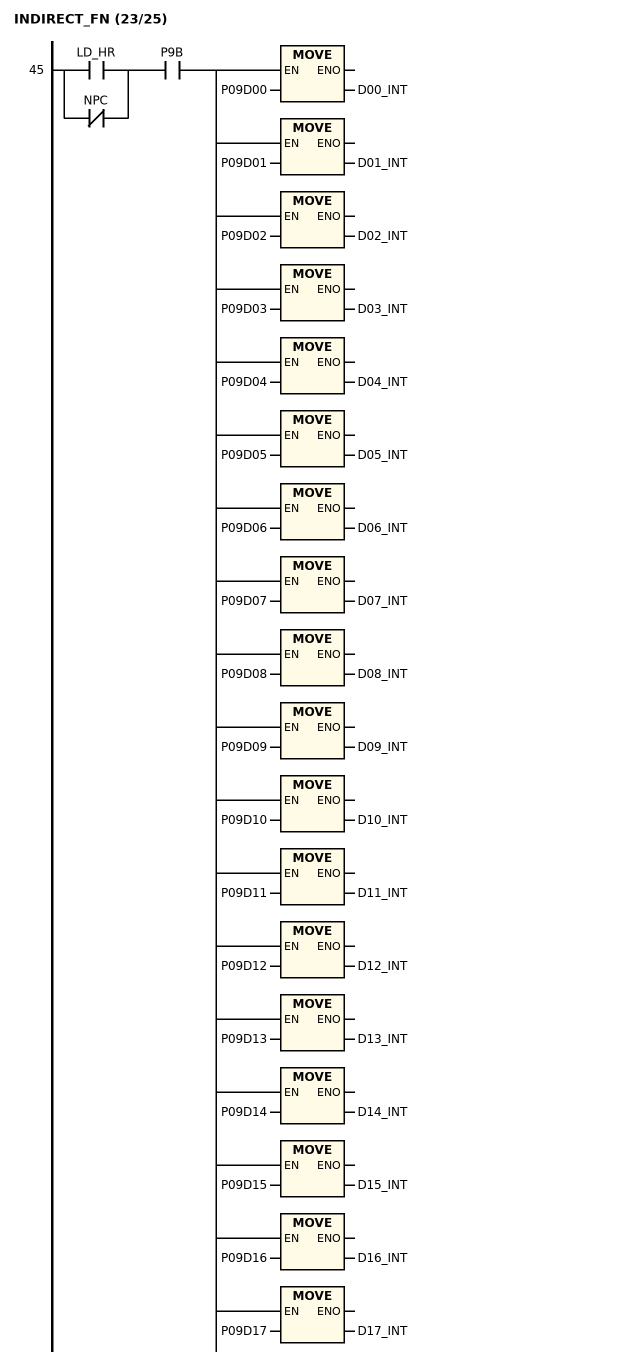
[picture p72: INDIRECT_FN (LD)]
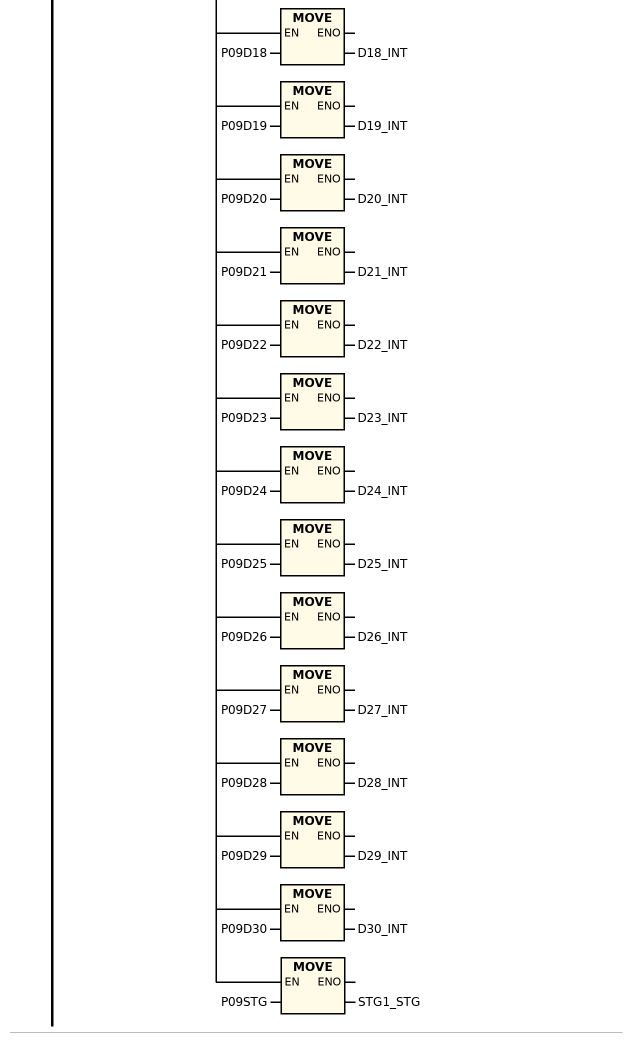
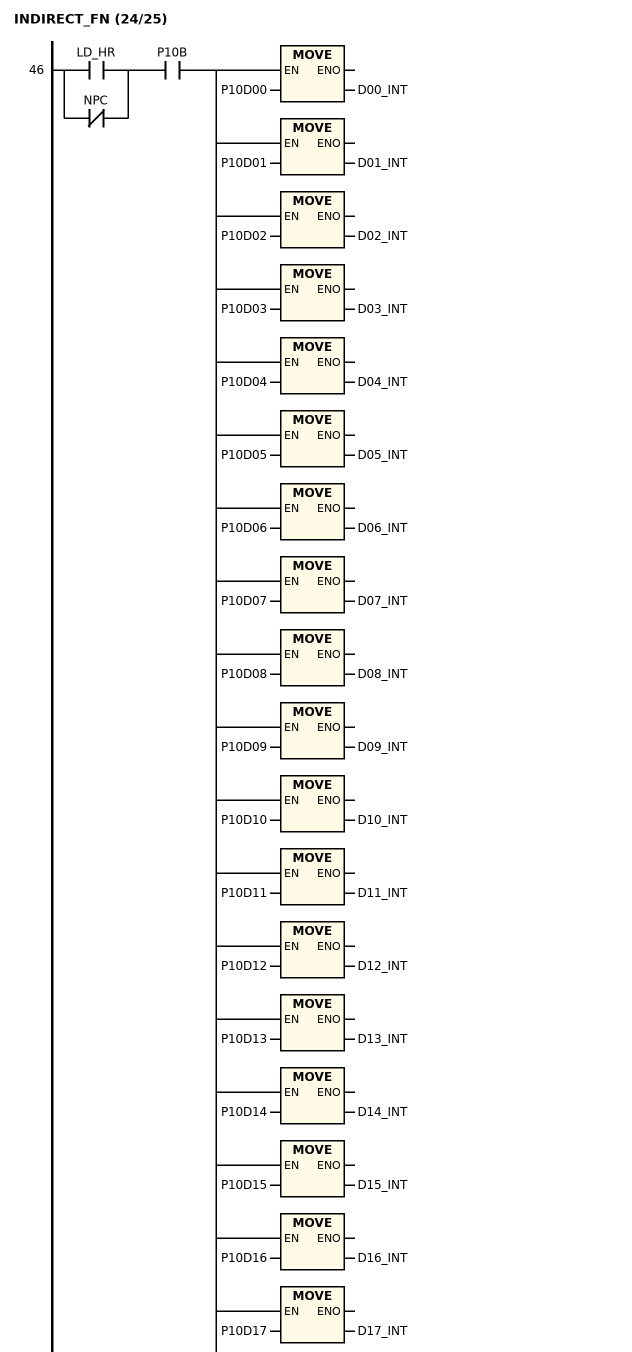
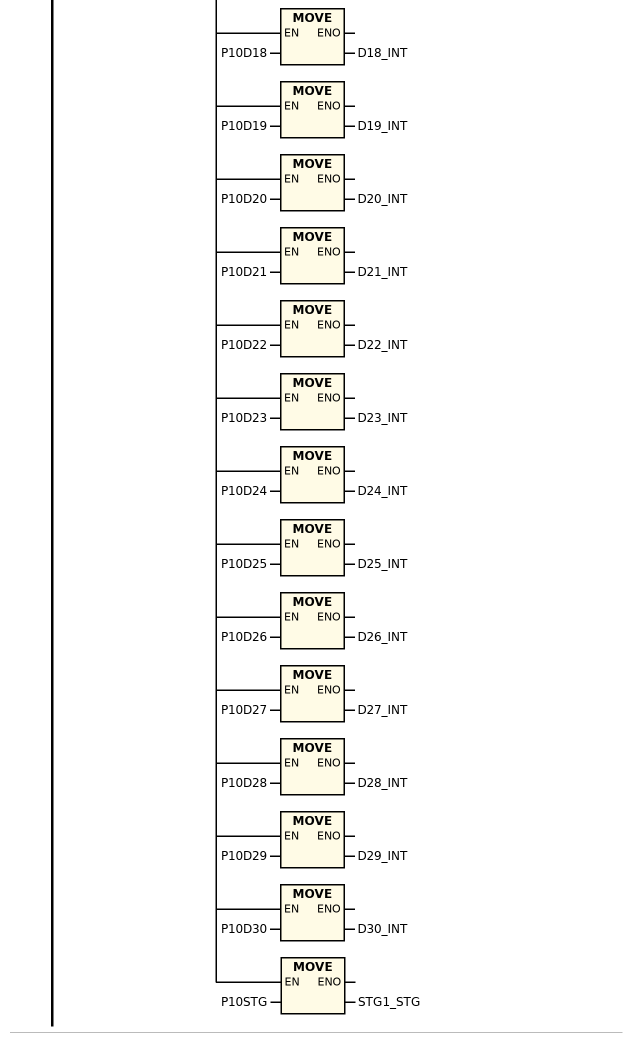
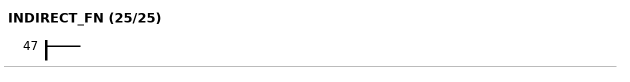
_LD_ (* Ladder Diagram *)
NETWORK 1
	[/LD_PB_IND_BOOL] - [NPC]
		EN --- MOVE(INT_D00) => D00_INT
		EN --- MOVE(INT_D01) => D01_INT
		EN --- MOVE(INT_D02) => D02_INT
		EN --- MOVE(INT_D03) => D03_INT
		EN --- MOVE(INT_D04) => D04_INT
		EN --- MOVE(INT_D05) => D05_INT
		EN --- MOVE(INT_D06) => D06_INT
		EN --- MOVE(INT_D07) => D07_INT
		EN --- MOVE(INT_D08) => D08_INT
		EN --- MOVE(INT_D09) => D09_INT
		EN --- MOVE(INT_D10) => D10_INT
		EN --- MOVE(INT_D11) => D11_INT
		EN --- MOVE(INT_D12) => D12_INT
		EN --- MOVE(INT_D13) => D13_INT
		EN --- MOVE(INT_D14) => D14_INT
		EN --- MOVE(INT_D15) => D15_INT
		EN --- MOVE(INT_D16) => D16_INT
		EN --- MOVE(INT_D17) => D17_INT
		EN --- MOVE(INT_D18) => D18_INT
		EN --- MOVE(INT_D19) => D19_INT
		EN --- MOVE(INT_D20) => D20_INT
		EN --- MOVE(INT_D21) => D21_INT
		EN --- MOVE(INT_D22) => D22_INT
		EN --- MOVE(INT_D23) => D23_INT
		EN --- MOVE(INT_D24) => D24_INT
		EN --- MOVE(INT_D25) => D25_INT
		EN --- MOVE(INT_D26) => D26_INT
		EN --- MOVE(INT_D27) => D27_INT
		EN --- MOVE(INT_D28) => D28_INT
		EN --- MOVE(INT_D29) => D29_INT
		EN --- MOVE(INT_D30) => D30_INT
		EN --- MOVE(STG_STG1) => STG1_STG
NETWORK 2
	*
		EN --- EQ(INT_P_NO, 1) => P1B
NETWORK 3
	*
		EN --- EQ(INT_P_NO, 2) => P2B
NETWORK 4
	*
		EN --- EQ(INT_P_NO, 3) => P3B
NETWORK 5
	*
		EN --- EQ(INT_P_NO, 4) => P4B
NETWORK 6
	*
		EN --- EQ(INT_P_NO, 5) => P5B
NETWORK 7
	*
		EN --- EQ(INT_P_NO, 6) => P6B
NETWORK 8
	*
		EN --- EQ(INT_P_NO, 7) => P7B
NETWORK 9
	*
		EN --- EQ(INT_P_NO, 8) => P8B
NETWORK 10
	*
		EN --- EQ(INT_P_NO, 9) => P9B
NETWORK 11
	*
		EN --- EQ(INT_P_NO, 10) => P10B
NETWORK 12
	[/N1] - TPC:TON(IN: *, PT: T#300ms) --- (N0)
NETWORK 13
	[N0] - TPC1:TON(IN: *, PT: T#100ms) --- (N1)
NETWORK 14
	[N0] - PCDF:R_TRIG(CLK: *) --- (PCTDF)
NETWORK 15
	[PCTDF]
		EN --- MOVE(INT_P_NO) => CNG_P_NO
NETWORK 16
	*
		EN --- EQ(INT_P_NO, CNG_P_NO) => NPC
NETWORK 17
	[BOOL_SV_PB] - SVPLS:R_TRIG(CLK: *) --- (SV_PB_PLS)
NETWORK 18
	{ [SV_PB_PLS] | [SV_HR] } - [/SV_CR] --- (SV_HR)
NETWORK 19
	[SV_HR] - SV_T:TON(IN: *, PT: T#1s) --- (SV_CR)
NETWORK 20
	[SV_HR] --- (SV_PB_IND_BOOL)
NETWORK 21
	[SV_HR] - SV_DF:R_TRIG(CLK: *) --- (SV_PLS)
NETWORK 22
	[SV_HR] - [P1B]
		EN --- MOVE(INT_D00) => P01D00
		EN --- MOVE(INT_D01) => P01D01
		EN --- MOVE(INT_D02) => P01D02
		EN --- MOVE(INT_D03) => P01D03
		EN --- MOVE(INT_D04) => P01D04
		EN --- MOVE(INT_D05) => P01D05
		EN --- MOVE(INT_D06) => P01D06
		EN --- MOVE(INT_D07) => P01D07
		EN --- MOVE(INT_D08) => P01D08
		EN --- MOVE(INT_D09) => P01D09
		EN --- MOVE(INT_D10) => P01D10
		EN --- MOVE(INT_D11) => P01D11
		EN --- MOVE(INT_D12) => P01D12
		EN --- MOVE(INT_D13) => P01D13
		EN --- MOVE(INT_D14) => P01D14
		EN --- MOVE(INT_D15) => P01D15
		EN --- MOVE(INT_D16) => P01D16
		EN --- MOVE(INT_D17) => P01D17
		EN --- MOVE(INT_D18) => P01D18
		EN --- MOVE(INT_D19) => P01D19
		EN --- MOVE(INT_D20) => P01D20
		EN --- MOVE(INT_D21) => P01D21
		EN --- MOVE(INT_D22) => P01D22
		EN --- MOVE(INT_D23) => P01D23
		EN --- MOVE(INT_D24) => P01D24
		EN --- MOVE(INT_D25) => P01D25
		EN --- MOVE(INT_D26) => P01D26
		EN --- MOVE(INT_D27) => P01D27
		EN --- MOVE(INT_D28) => P01D28
		EN --- MOVE(INT_D29) => P01D29
		EN --- MOVE(INT_D30) => P01D30
		EN --- MOVE(STG_STG1) => P01STG
NETWORK 23
	[SV_HR] - [P2B]
		EN --- MOVE(INT_D00) => P02D00
		EN --- MOVE(INT_D01) => P02D01
		EN --- MOVE(INT_D02) => P02D02
		EN --- MOVE(INT_D03) => P02D03
		EN --- MOVE(INT_D04) => P02D04
		EN --- MOVE(INT_D05) => P02D05
		EN --- MOVE(INT_D06) => P02D06
		EN --- MOVE(INT_D07) => P02D07
		EN --- MOVE(INT_D08) => P02D08
		EN --- MOVE(INT_D09) => P02D09
		EN --- MOVE(INT_D10) => P02D10
		EN --- MOVE(INT_D11) => P02D11
		EN --- MOVE(INT_D12) => P02D12
		EN --- MOVE(INT_D13) => P02D13
		EN --- MOVE(INT_D14) => P02D14
		EN --- MOVE(INT_D15) => P02D15
		EN --- MOVE(INT_D16) => P02D16
		EN --- MOVE(INT_D17) => P02D17
		EN --- MOVE(INT_D18) => P02D18
		EN --- MOVE(INT_D19) => P02D19
		EN --- MOVE(INT_D20) => P02D20
		EN --- MOVE(INT_D21) => P02D21
		EN --- MOVE(INT_D22) => P02D22
		EN --- MOVE(INT_D23) => P02D23
		EN --- MOVE(INT_D24) => P02D24
		EN --- MOVE(INT_D25) => P02D25
		EN --- MOVE(INT_D26) => P02D26
		EN --- MOVE(INT_D27) => P02D27
		EN --- MOVE(INT_D28) => P02D28
		EN --- MOVE(INT_D29) => P02D29
		EN --- MOVE(INT_D30) => P02D30
		EN --- MOVE(STG_STG1) => P02STG
NETWORK 24
	[SV_HR] - [P3B]
		EN --- MOVE(INT_D00) => P03D00
		EN --- MOVE(INT_D01) => P03D01
		EN --- MOVE(INT_D02) => P03D02
		EN --- MOVE(INT_D03) => P03D03
		EN --- MOVE(INT_D04) => P03D04
		EN --- MOVE(INT_D05) => P03D05
		EN --- MOVE(INT_D06) => P03D06
		EN --- MOVE(INT_D07) => P03D07
		EN --- MOVE(INT_D08) => P03D08
		EN --- MOVE(INT_D09) => P03D09
		EN --- MOVE(INT_D10) => P03D10
		EN --- MOVE(INT_D11) => P03D11
		EN --- MOVE(INT_D12) => P03D12
		EN --- MOVE(INT_D13) => P03D13
		EN --- MOVE(INT_D14) => P03D14
		EN --- MOVE(INT_D15) => P03D15
		EN --- MOVE(INT_D16) => P03D16
		EN --- MOVE(INT_D17) => P03D17
		EN --- MOVE(INT_D18) => P03D18
		EN --- MOVE(INT_D19) => P03D19
		EN --- MOVE(INT_D20) => P03D20
		EN --- MOVE(INT_D21) => P03D21
		EN --- MOVE(INT_D22) => P03D22
		EN --- MOVE(INT_D23) => P03D23
		EN --- MOVE(INT_D24) => P03D24
		EN --- MOVE(INT_D25) => P03D25
		EN --- MOVE(INT_D26) => P03D26
		EN --- MOVE(INT_D27) => P03D27
		EN --- MOVE(INT_D28) => P03D28
		EN --- MOVE(INT_D29) => P03D29
		EN --- MOVE(INT_D30) => P03D30
		EN --- MOVE(STG_STG1) => P03STG
NETWORK 25
	[SV_HR] - [P4B]
		EN --- MOVE(INT_D00) => P04D00
		EN --- MOVE(INT_D01) => P04D01
		EN --- MOVE(INT_D02) => P04D02
		EN --- MOVE(INT_D03) => P04D03
		EN --- MOVE(INT_D04) => P04D04
		EN --- MOVE(INT_D05) => P04D05
		EN --- MOVE(INT_D06) => P04D06
		EN --- MOVE(INT_D07) => P04D07
		EN --- MOVE(INT_D08) => P04D08
		EN --- MOVE(INT_D09) => P04D09
		EN --- MOVE(INT_D10) => P04D10
		EN --- MOVE(INT_D11) => P04D11
		EN --- MOVE(INT_D12) => P04D12
		EN --- MOVE(INT_D13) => P04D13
		EN --- MOVE(INT_D14) => P04D14
		EN --- MOVE(INT_D15) => P04D15
		EN --- MOVE(INT_D16) => P04D16
		EN --- MOVE(INT_D17) => P04D17
		EN --- MOVE(INT_D18) => P04D18
		EN --- MOVE(INT_D19) => P04D19
		EN --- MOVE(INT_D20) => P04D20
		EN --- MOVE(INT_D21) => P04D21
		EN --- MOVE(INT_D22) => P04D22
		EN --- MOVE(INT_D23) => P04D23
		EN --- MOVE(INT_D24) => P04D24
		EN --- MOVE(INT_D25) => P04D25
		EN --- MOVE(INT_D26) => P04D26
		EN --- MOVE(INT_D27) => P04D27
		EN --- MOVE(INT_D28) => P04D28
		EN --- MOVE(INT_D29) => P04D29
		EN --- MOVE(INT_D30) => P04D30
		EN --- MOVE(STG_STG1) => P04STG
NETWORK 26
	[SV_HR] - [P5B]
		EN --- MOVE(INT_D00) => P05D00
		EN --- MOVE(INT_D01) => P05D01
		EN --- MOVE(INT_D02) => P05D02
		EN --- MOVE(INT_D03) => P05D03
		EN --- MOVE(INT_D04) => P05D04
		EN --- MOVE(INT_D05) => P05D05
		EN --- MOVE(INT_D06) => P05D06
		EN --- MOVE(INT_D07) => P05D07
		EN --- MOVE(INT_D08) => P05D08
		EN --- MOVE(INT_D09) => P05D09
		EN --- MOVE(INT_D10) => P05D10
		EN --- MOVE(INT_D11) => P05D11
		EN --- MOVE(INT_D12) => P05D12
		EN --- MOVE(INT_D13) => P05D13
		EN --- MOVE(INT_D14) => P05D14
		EN --- MOVE(INT_D15) => P05D15
		EN --- MOVE(INT_D16) => P05D16
		EN --- MOVE(INT_D17) => P05D17
		EN --- MOVE(INT_D18) => P05D18
		EN --- MOVE(INT_D19) => P05D19
		EN --- MOVE(INT_D20) => P05D20
		EN --- MOVE(INT_D21) => P05D21
		EN --- MOVE(INT_D22) => P05D22
		EN --- MOVE(INT_D23) => P05D23
		EN --- MOVE(INT_D24) => P05D24
		EN --- MOVE(INT_D25) => P05D25
		EN --- MOVE(INT_D26) => P05D26
		EN --- MOVE(INT_D27) => P05D27
		EN --- MOVE(INT_D28) => P05D28
		EN --- MOVE(INT_D29) => P05D29
		EN --- MOVE(INT_D30) => P05D30
		EN --- MOVE(STG_STG1) => P05STG
NETWORK 27
	[SV_HR] - [P6B]
		EN --- MOVE(INT_D00) => P06D00
		EN --- MOVE(INT_D01) => P06D01
		EN --- MOVE(INT_D02) => P06D02
		EN --- MOVE(INT_D03) => P06D03
		EN --- MOVE(INT_D04) => P06D04
		EN --- MOVE(INT_D05) => P06D05
		EN --- MOVE(INT_D06) => P06D06
		EN --- MOVE(INT_D07) => P06D07
		EN --- MOVE(INT_D08) => P06D08
		EN --- MOVE(INT_D09) => P06D09
		EN --- MOVE(INT_D10) => P06D10
		EN --- MOVE(INT_D11) => P06D11
		EN --- MOVE(INT_D12) => P06D12
		EN --- MOVE(INT_D13) => P06D13
		EN --- MOVE(INT_D14) => P06D14
		EN --- MOVE(INT_D15) => P06D15
		EN --- MOVE(INT_D16) => P06D16
		EN --- MOVE(INT_D17) => P06D17
		EN --- MOVE(INT_D18) => P06D18
		EN --- MOVE(INT_D19) => P06D19
		EN --- MOVE(INT_D20) => P06D20
		EN --- MOVE(INT_D21) => P06D21
		EN --- MOVE(INT_D22) => P06D22
		EN --- MOVE(INT_D23) => P06D23
		EN --- MOVE(INT_D24) => P06D24
		EN --- MOVE(INT_D25) => P06D25
		EN --- MOVE(INT_D26) => P06D26
		EN --- MOVE(INT_D27) => P06D27
		EN --- MOVE(INT_D28) => P06D28
		EN --- MOVE(INT_D29) => P06D29
		EN --- MOVE(INT_D30) => P06D30
		EN --- MOVE(STG_STG1) => P06STG
NETWORK 28
	[SV_HR] - [P7B]
		EN --- MOVE(INT_D00) => P07D00
		EN --- MOVE(INT_D01) => P07D01
		EN --- MOVE(INT_D02) => P07D02
		EN --- MOVE(INT_D03) => P07D03
		EN --- MOVE(INT_D04) => P07D04
		EN --- MOVE(INT_D05) => P07D05
		EN --- MOVE(INT_D06) => P07D06
		EN --- MOVE(INT_D07) => P07D07
		EN --- MOVE(INT_D08) => P07D08
		EN --- MOVE(INT_D09) => P07D09
		EN --- MOVE(INT_D10) => P07D10
		EN --- MOVE(INT_D11) => P07D11
		EN --- MOVE(INT_D12) => P07D12
		EN --- MOVE(INT_D13) => P07D13
		EN --- MOVE(INT_D14) => P07D14
		EN --- MOVE(INT_D15) => P07D15
		EN --- MOVE(INT_D16) => P07D16
		EN --- MOVE(INT_D17) => P07D17
		EN --- MOVE(INT_D18) => P07D18
		EN --- MOVE(INT_D19) => P07D19
		EN --- MOVE(INT_D20) => P07D20
		EN --- MOVE(INT_D21) => P07D21
		EN --- MOVE(INT_D22) => P07D22
		EN --- MOVE(INT_D23) => P07D23
		EN --- MOVE(INT_D24) => P07D24
		EN --- MOVE(INT_D25) => P07D25
		EN --- MOVE(INT_D26) => P07D26
		EN --- MOVE(INT_D27) => P07D27
		EN --- MOVE(INT_D28) => P07D28
		EN --- MOVE(INT_D29) => P07D29
		EN --- MOVE(INT_D30) => P07D30
		EN --- MOVE(STG_STG1) => P07STG
NETWORK 29
	[SV_HR] - [P8B]
		EN --- MOVE(INT_D00) => P08D00
		EN --- MOVE(INT_D01) => P08D01
		EN --- MOVE(INT_D02) => P08D02
		EN --- MOVE(INT_D03) => P08D03
		EN --- MOVE(INT_D04) => P08D04
		EN --- MOVE(INT_D05) => P08D05
		EN --- MOVE(INT_D06) => P08D06
		EN --- MOVE(INT_D07) => P08D07
		EN --- MOVE(INT_D08) => P08D08
		EN --- MOVE(INT_D09) => P08D09
		EN --- MOVE(INT_D10) => P08D10
		EN --- MOVE(INT_D11) => P08D11
		EN --- MOVE(INT_D12) => P08D12
		EN --- MOVE(INT_D13) => P08D13
		EN --- MOVE(INT_D14) => P08D14
		EN --- MOVE(INT_D15) => P08D15
		EN --- MOVE(INT_D16) => P08D16
		EN --- MOVE(INT_D17) => P08D17
		EN --- MOVE(INT_D18) => P08D18
		EN --- MOVE(INT_D19) => P08D19
		EN --- MOVE(INT_D20) => P08D20
		EN --- MOVE(INT_D21) => P08D21
		EN --- MOVE(INT_D22) => P08D22
		EN --- MOVE(INT_D23) => P08D23
		EN --- MOVE(INT_D24) => P08D24
		EN --- MOVE(INT_D25) => P08D25
		EN --- MOVE(INT_D26) => P08D26
		EN --- MOVE(INT_D27) => P08D27
		EN --- MOVE(INT_D28) => P08D28
		EN --- MOVE(INT_D29) => P08D29
		EN --- MOVE(INT_D30) => P08D30
		EN --- MOVE(STG_STG1) => P08STG
NETWORK 30
	[SV_HR] - [P9B]
		EN --- MOVE(INT_D00) => P09D00
		EN --- MOVE(INT_D01) => P09D01
		EN --- MOVE(INT_D02) => P09D02
		EN --- MOVE(INT_D03) => P09D03
		EN --- MOVE(INT_D04) => P09D04
		EN --- MOVE(INT_D05) => P09D05
		EN --- MOVE(INT_D06) => P09D06
		EN --- MOVE(INT_D07) => P09D07
		EN --- MOVE(INT_D08) => P09D08
		EN --- MOVE(INT_D09) => P09D09
		EN --- MOVE(INT_D10) => P09D10
		EN --- MOVE(INT_D11) => P09D11
		EN --- MOVE(INT_D12) => P09D12
		EN --- MOVE(INT_D13) => P09D13
		EN --- MOVE(INT_D14) => P09D14
		EN --- MOVE(INT_D15) => P09D15
		EN --- MOVE(INT_D16) => P09D16
		EN --- MOVE(INT_D17) => P09D17
		EN --- MOVE(INT_D18) => P09D18
		EN --- MOVE(INT_D19) => P09D19
		EN --- MOVE(INT_D20) => P09D20
		EN --- MOVE(INT_D21) => P09D21
		EN --- MOVE(INT_D22) => P09D22
		EN --- MOVE(INT_D23) => P09D23
		EN --- MOVE(INT_D24) => P09D24
		EN --- MOVE(INT_D25) => P09D25
		EN --- MOVE(INT_D26) => P09D26
		EN --- MOVE(INT_D27) => P09D27
		EN --- MOVE(INT_D28) => P09D28
		EN --- MOVE(INT_D29) => P09D29
		EN --- MOVE(INT_D30) => P09D30
		EN --- MOVE(STG_STG1) => P09STG
NETWORK 31
	[SV_HR] - [P10B]
		EN --- MOVE(INT_D00) => P10D00
		EN --- MOVE(INT_D01) => P10D01
		EN --- MOVE(INT_D02) => P10D02
		EN --- MOVE(INT_D03) => P10D03
		EN --- MOVE(INT_D04) => P10D04
		EN --- MOVE(INT_D05) => P10D05
		EN --- MOVE(INT_D06) => P10D06
		EN --- MOVE(INT_D07) => P10D07
		EN --- MOVE(INT_D08) => P10D08
		EN --- MOVE(INT_D09) => P10D09
		EN --- MOVE(INT_D10) => P10D10
		EN --- MOVE(INT_D11) => P10D11
		EN --- MOVE(INT_D12) => P10D12
		EN --- MOVE(INT_D13) => P10D13
		EN --- MOVE(INT_D14) => P10D14
		EN --- MOVE(INT_D15) => P10D15
		EN --- MOVE(INT_D16) => P10D16
		EN --- MOVE(INT_D17) => P10D17
		EN --- MOVE(INT_D18) => P10D18
		EN --- MOVE(INT_D19) => P10D19
		EN --- MOVE(INT_D20) => P10D20
		EN --- MOVE(INT_D21) => P10D21
		EN --- MOVE(INT_D22) => P10D22
		EN --- MOVE(INT_D23) => P10D23
		EN --- MOVE(INT_D24) => P10D24
		EN --- MOVE(INT_D25) => P10D25
		EN --- MOVE(INT_D26) => P10D26
		EN --- MOVE(INT_D27) => P10D27
		EN --- MOVE(INT_D28) => P10D28
		EN --- MOVE(INT_D29) => P10D29
		EN --- MOVE(INT_D30) => P10D30
		EN --- MOVE(STG_STG1) => P10STG
NETWORK 32
	[BOOL_LD_PB] - LDPLS:R_TRIG(CLK: *) --- (LD_PB_PLS)
NETWORK 33
	{ [LD_PB_PLS] | [LD_HR] } - [/LD_CR] --- (LD_HR)
NETWORK 34
	[LD_HR] - LD_T:TON(IN: *, PT: T#1s) --- (LD_CR)
NETWORK 35
	[LD_HR] --- (LD_PB_IND_BOOL)
NETWORK 36
	[LD_HR] - LD_DF:R_TRIG(CLK: *) --- (LD_PLS)
NETWORK 37
	{ [LD_HR] | [/NPC] } - [P1B]
		EN --- MOVE(P01D00) => D00_INT
		EN --- MOVE(P01D01) => D01_INT
		EN --- MOVE(P01D02) => D02_INT
		EN --- MOVE(P01D03) => D03_INT
		EN --- MOVE(P01D04) => D04_INT
		EN --- MOVE(P01D05) => D05_INT
		EN --- MOVE(P01D06) => D06_INT
		EN --- MOVE(P01D07) => D07_INT
		EN --- MOVE(P01D08) => D08_INT
		EN --- MOVE(P01D09) => D09_INT
		EN --- MOVE(P01D10) => D10_INT
		EN --- MOVE(P01D11) => D11_INT
		EN --- MOVE(P01D12) => D12_INT
		EN --- MOVE(P01D13) => D13_INT
		EN --- MOVE(P01D14) => D14_INT
		EN --- MOVE(P01D15) => D15_INT
		EN --- MOVE(P01D16) => D16_INT
		EN --- MOVE(P01D17) => D17_INT
		EN --- MOVE(P01D18) => D18_INT
		EN --- MOVE(P01D19) => D19_INT
		EN --- MOVE(P01D20) => D20_INT
		EN --- MOVE(P01D21) => D21_INT
		EN --- MOVE(P01D22) => D22_INT
		EN --- MOVE(P01D23) => D23_INT
		EN --- MOVE(P01D24) => D24_INT
		EN --- MOVE(P01D25) => D25_INT
		EN --- MOVE(P01D26) => D26_INT
		EN --- MOVE(P01D27) => D27_INT
		EN --- MOVE(P01D28) => D28_INT
		EN --- MOVE(P01D29) => D29_INT
		EN --- MOVE(P01D30) => D30_INT
		EN --- MOVE(P01STG) => STG1_STG
NETWORK 38
	{ [LD_HR] | [/NPC] } - [P2B]
		EN --- MOVE(P02D00) => D00_INT
		EN --- MOVE(P02D01) => D01_INT
		EN --- MOVE(P02D02) => D02_INT
		EN --- MOVE(P02D03) => D03_INT
		EN --- MOVE(P02D04) => D04_INT
		EN --- MOVE(P02D05) => D05_INT
		EN --- MOVE(P02D06) => D06_INT
		EN --- MOVE(P02D07) => D07_INT
		EN --- MOVE(P02D08) => D08_INT
		EN --- MOVE(P02D09) => D09_INT
		EN --- MOVE(P02D10) => D10_INT
		EN --- MOVE(P02D11) => D11_INT
		EN --- MOVE(P02D12) => D12_INT
		EN --- MOVE(P02D13) => D13_INT
		EN --- MOVE(P02D14) => D14_INT
		EN --- MOVE(P02D15) => D15_INT
		EN --- MOVE(P02D16) => D16_INT
		EN --- MOVE(P02D17) => D17_INT
		EN --- MOVE(P02D18) => D18_INT
		EN --- MOVE(P02D19) => D19_INT
		EN --- MOVE(P02D20) => D20_INT
		EN --- MOVE(P02D21) => D21_INT
		EN --- MOVE(P02D22) => D22_INT
		EN --- MOVE(P02D23) => D23_INT
		EN --- MOVE(P02D24) => D24_INT
		EN --- MOVE(P02D25) => D25_INT
		EN --- MOVE(P02D26) => D26_INT
		EN --- MOVE(P02D27) => D27_INT
		EN --- MOVE(P02D28) => D28_INT
		EN --- MOVE(P02D29) => D29_INT
		EN --- MOVE(P02D30) => D30_INT
		EN --- MOVE(P02STG) => STG1_STG
NETWORK 39
	{ [LD_HR] | [/NPC] } - [P3B]
		EN --- MOVE(P03D00) => D00_INT
		EN --- MOVE(P03D01) => D01_INT
		EN --- MOVE(P03D02) => D02_INT
		EN --- MOVE(P03D03) => D03_INT
		EN --- MOVE(P03D04) => D04_INT
		EN --- MOVE(P03D05) => D05_INT
		EN --- MOVE(P03D06) => D06_INT
		EN --- MOVE(P03D07) => D07_INT
		EN --- MOVE(P03D08) => D08_INT
		EN --- MOVE(P03D09) => D09_INT
		EN --- MOVE(P03D10) => D10_INT
		EN --- MOVE(P03D11) => D11_INT
		EN --- MOVE(P03D12) => D12_INT
		EN --- MOVE(P03D13) => D13_INT
		EN --- MOVE(P03D14) => D14_INT
		EN --- MOVE(P03D15) => D15_INT
		EN --- MOVE(P03D16) => D16_INT
		EN --- MOVE(P03D17) => D17_INT
		EN --- MOVE(P03D18) => D18_INT
		EN --- MOVE(P03D19) => D19_INT
		EN --- MOVE(P03D20) => D20_INT
		EN --- MOVE(P03D21) => D21_INT
		EN --- MOVE(P03D22) => D22_INT
		EN --- MOVE(P03D23) => D23_INT
		EN --- MOVE(P03D24) => D24_INT
		EN --- MOVE(P03D25) => D25_INT
		EN --- MOVE(P03D26) => D26_INT
		EN --- MOVE(P03D27) => D27_INT
		EN --- MOVE(P03D28) => D28_INT
		EN --- MOVE(P03D29) => D29_INT
		EN --- MOVE(P03D30) => D30_INT
		EN --- MOVE(P03STG) => STG1_STG
NETWORK 40
	{ [LD_HR] | [/NPC] } - [P4B]
		EN --- MOVE(P04D00) => D00_INT
		EN --- MOVE(P04D01) => D01_INT
		EN --- MOVE(P04D02) => D02_INT
		EN --- MOVE(P04D03) => D03_INT
		EN --- MOVE(P04D04) => D04_INT
		EN --- MOVE(P04D05) => D05_INT
		EN --- MOVE(P04D06) => D06_INT
		EN --- MOVE(P04D07) => D07_INT
		EN --- MOVE(P04D08) => D08_INT
		EN --- MOVE(P04D09) => D09_INT
		EN --- MOVE(P04D10) => D10_INT
		EN --- MOVE(P04D11) => D11_INT
		EN --- MOVE(P04D12) => D12_INT
		EN --- MOVE(P04D13) => D13_INT
		EN --- MOVE(P04D14) => D14_INT
		EN --- MOVE(P04D15) => D15_INT
		EN --- MOVE(P04D16) => D16_INT
		EN --- MOVE(P04D17) => D17_INT
		EN --- MOVE(P04D18) => D18_INT
		EN --- MOVE(P04D19) => D19_INT
		EN --- MOVE(P04D20) => D20_INT
		EN --- MOVE(P04D21) => D21_INT
		EN --- MOVE(P04D22) => D22_INT
		EN --- MOVE(P04D23) => D23_INT
		EN --- MOVE(P04D24) => D24_INT
		EN --- MOVE(P04D25) => D25_INT
		EN --- MOVE(P04D26) => D26_INT
		EN --- MOVE(P04D27) => D27_INT
		EN --- MOVE(P04D28) => D28_INT
		EN --- MOVE(P04D29) => D29_INT
		EN --- MOVE(P04D30) => D30_INT
		EN --- MOVE(P04STG) => STG1_STG
NETWORK 41
	{ [LD_HR] | [/NPC] } - [P5B]
		EN --- MOVE(P05D00) => D00_INT
		EN --- MOVE(P05D01) => D01_INT
		EN --- MOVE(P05D02) => D02_INT
		EN --- MOVE(P05D03) => D03_INT
		EN --- MOVE(P05D04) => D04_INT
		EN --- MOVE(P05D05) => D05_INT
		EN --- MOVE(P05D06) => D06_INT
		EN --- MOVE(P05D07) => D07_INT
		EN --- MOVE(P05D08) => D08_INT
		EN --- MOVE(P05D09) => D09_INT
		EN --- MOVE(P05D10) => D10_INT
		EN --- MOVE(P05D11) => D11_INT
		EN --- MOVE(P05D12) => D12_INT
		EN --- MOVE(P05D13) => D13_INT
		EN --- MOVE(P05D14) => D14_INT
		EN --- MOVE(P05D15) => D15_INT
		EN --- MOVE(P05D16) => D16_INT
		EN --- MOVE(P05D17) => D17_INT
		EN --- MOVE(P05D18) => D18_INT
		EN --- MOVE(P05D19) => D19_INT
		EN --- MOVE(P05D20) => D20_INT
		EN --- MOVE(P05D21) => D21_INT
		EN --- MOVE(P05D22) => D22_INT
		EN --- MOVE(P05D23) => D23_INT
		EN --- MOVE(P05D24) => D24_INT
		EN --- MOVE(P05D25) => D25_INT
		EN --- MOVE(P05D26) => D26_INT
		EN --- MOVE(P05D27) => D27_INT
		EN --- MOVE(P05D28) => D28_INT
		EN --- MOVE(P05D29) => D29_INT
		EN --- MOVE(P05D30) => D30_INT
		EN --- MOVE(P05STG) => STG1_STG
NETWORK 42
	{ [LD_HR] | [/NPC] } - [P6B]
		EN --- MOVE(P06D00) => D00_INT
		EN --- MOVE(P06D01) => D01_INT
		EN --- MOVE(P06D02) => D02_INT
		EN --- MOVE(P06D03) => D03_INT
		EN --- MOVE(P06D04) => D04_INT
		EN --- MOVE(P06D05) => D05_INT
		EN --- MOVE(P06D06) => D06_INT
		EN --- MOVE(P06D07) => D07_INT
		EN --- MOVE(P06D08) => D08_INT
		EN --- MOVE(P06D09) => D09_INT
		EN --- MOVE(P06D10) => D10_INT
		EN --- MOVE(P06D11) => D11_INT
		EN --- MOVE(P06D12) => D12_INT
		EN --- MOVE(P06D13) => D13_INT
		EN --- MOVE(P06D14) => D14_INT
		EN --- MOVE(P06D15) => D15_INT
		EN --- MOVE(P06D16) => D16_INT
		EN --- MOVE(P06D17) => D17_INT
		EN --- MOVE(P06D18) => D18_INT
		EN --- MOVE(P06D19) => D19_INT
		EN --- MOVE(P06D20) => D20_INT
		EN --- MOVE(P06D21) => D21_INT
		EN --- MOVE(P06D22) => D22_INT
		EN --- MOVE(P06D23) => D23_INT
		EN --- MOVE(P06D24) => D24_INT
		EN --- MOVE(P06D25) => D25_INT
		EN --- MOVE(P06D26) => D26_INT
		EN --- MOVE(P06D27) => D27_INT
		EN --- MOVE(P06D28) => D28_INT
		EN --- MOVE(P06D29) => D29_INT
		EN --- MOVE(P06D30) => D30_INT
		EN --- MOVE(P06STG) => STG1_STG
NETWORK 43
	{ [LD_HR] | [/NPC] } - [P7B]
		EN --- MOVE(P07D00) => D00_INT
		EN --- MOVE(P07D01) => D01_INT
		EN --- MOVE(P07D02) => D02_INT
		EN --- MOVE(P07D03) => D03_INT
		EN --- MOVE(P07D04) => D04_INT
		EN --- MOVE(P07D05) => D05_INT
		EN --- MOVE(P07D06) => D06_INT
		EN --- MOVE(P07D07) => D07_INT
		EN --- MOVE(P07D08) => D08_INT
		EN --- MOVE(P07D09) => D09_INT
		EN --- MOVE(P07D10) => D10_INT
		EN --- MOVE(P07D11) => D11_INT
		EN --- MOVE(P07D12) => D12_INT
		EN --- MOVE(P07D13) => D13_INT
		EN --- MOVE(P07D14) => D14_INT
		EN --- MOVE(P07D15) => D15_INT
		EN --- MOVE(P07D16) => D16_INT
		EN --- MOVE(P07D17) => D17_INT
		EN --- MOVE(P07D18) => D18_INT
		EN --- MOVE(P07D19) => D19_INT
		EN --- MOVE(P07D20) => D20_INT
		EN --- MOVE(P07D21) => D21_INT
		EN --- MOVE(P07D22) => D22_INT
		EN --- MOVE(P07D23) => D23_INT
		EN --- MOVE(P07D24) => D24_INT
		EN --- MOVE(P07D25) => D25_INT
		EN --- MOVE(P07D26) => D26_INT
		EN --- MOVE(P07D27) => D27_INT
		EN --- MOVE(P07D28) => D28_INT
		EN --- MOVE(P07D29) => D29_INT
		EN --- MOVE(P07D30) => D30_INT
		EN --- MOVE(P07STG) => STG1_STG
NETWORK 44
	{ [LD_HR] | [/NPC] } - [P8B]
		EN --- MOVE(P08D00) => D00_INT
		EN --- MOVE(P08D01) => D01_INT
		EN --- MOVE(P08D02) => D02_INT
		EN --- MOVE(P08D03) => D03_INT
		EN --- MOVE(P08D04) => D04_INT
		EN --- MOVE(P08D05) => D05_INT
		EN --- MOVE(P08D06) => D06_INT
		EN --- MOVE(P08D07) => D07_INT
		EN --- MOVE(P08D08) => D08_INT
		EN --- MOVE(P08D09) => D09_INT
		EN --- MOVE(P08D10) => D10_INT
		EN --- MOVE(P08D11) => D11_INT
		EN --- MOVE(P08D12) => D12_INT
		EN --- MOVE(P08D13) => D13_INT
		EN --- MOVE(P08D14) => D14_INT
		EN --- MOVE(P08D15) => D15_INT
		EN --- MOVE(P08D16) => D16_INT
		EN --- MOVE(P08D17) => D17_INT
		EN --- MOVE(P08D18) => D18_INT
		EN --- MOVE(P08D19) => D19_INT
		EN --- MOVE(P08D20) => D20_INT
		EN --- MOVE(P08D21) => D21_INT
		EN --- MOVE(P08D22) => D22_INT
		EN --- MOVE(P08D23) => D23_INT
		EN --- MOVE(P08D24) => D24_INT
		EN --- MOVE(P08D25) => D25_INT
		EN --- MOVE(P08D26) => D26_INT
		EN --- MOVE(P08D27) => D27_INT
		EN --- MOVE(P08D28) => D28_INT
		EN --- MOVE(P08D29) => D29_INT
		EN --- MOVE(P08D30) => D30_INT
		EN --- MOVE(P08STG) => STG1_STG
NETWORK 45
	{ [LD_HR] | [/NPC] } - [P9B]
		EN --- MOVE(P09D00) => D00_INT
		EN --- MOVE(P09D01) => D01_INT
		EN --- MOVE(P09D02) => D02_INT
		EN --- MOVE(P09D03) => D03_INT
		EN --- MOVE(P09D04) => D04_INT
		EN --- MOVE(P09D05) => D05_INT
		EN --- MOVE(P09D06) => D06_INT
		EN --- MOVE(P09D07) => D07_INT
		EN --- MOVE(P09D08) => D08_INT
		EN --- MOVE(P09D09) => D09_INT
		EN --- MOVE(P09D10) => D10_INT
		EN --- MOVE(P09D11) => D11_INT
		EN --- MOVE(P09D12) => D12_INT
		EN --- MOVE(P09D13) => D13_INT
		EN --- MOVE(P09D14) => D14_INT
		EN --- MOVE(P09D15) => D15_INT
		EN --- MOVE(P09D16) => D16_INT
		EN --- MOVE(P09D17) => D17_INT
		EN --- MOVE(P09D18) => D18_INT
		EN --- MOVE(P09D19) => D19_INT
		EN --- MOVE(P09D20) => D20_INT
		EN --- MOVE(P09D21) => D21_INT
		EN --- MOVE(P09D22) => D22_INT
		EN --- MOVE(P09D23) => D23_INT
		EN --- MOVE(P09D24) => D24_INT
		EN --- MOVE(P09D25) => D25_INT
		EN --- MOVE(P09D26) => D26_INT
		EN --- MOVE(P09D27) => D27_INT
		EN --- MOVE(P09D28) => D28_INT
		EN --- MOVE(P09D29) => D29_INT
		EN --- MOVE(P09D30) => D30_INT
		EN --- MOVE(P09STG) => STG1_STG
NETWORK 46
	{ [LD_HR] | [/NPC] } - [P10B]
		EN --- MOVE(P10D00) => D00_INT
		EN --- MOVE(P10D01) => D01_INT
		EN --- MOVE(P10D02) => D02_INT
		EN --- MOVE(P10D03) => D03_INT
		EN --- MOVE(P10D04) => D04_INT
		EN --- MOVE(P10D05) => D05_INT
		EN --- MOVE(P10D06) => D06_INT
		EN --- MOVE(P10D07) => D07_INT
		EN --- MOVE(P10D08) => D08_INT
		EN --- MOVE(P10D09) => D09_INT
		EN --- MOVE(P10D10) => D10_INT
		EN --- MOVE(P10D11) => D11_INT
		EN --- MOVE(P10D12) => D12_INT
		EN --- MOVE(P10D13) => D13_INT
		EN --- MOVE(P10D14) => D14_INT
		EN --- MOVE(P10D15) => D15_INT
		EN --- MOVE(P10D16) => D16_INT
		EN --- MOVE(P10D17) => D17_INT
		EN --- MOVE(P10D18) => D18_INT
		EN --- MOVE(P10D19) => D19_INT
		EN --- MOVE(P10D20) => D20_INT
		EN --- MOVE(P10D21) => D21_INT
		EN --- MOVE(P10D22) => D22_INT
		EN --- MOVE(P10D23) => D23_INT
		EN --- MOVE(P10D24) => D24_INT
		EN --- MOVE(P10D25) => D25_INT
		EN --- MOVE(P10D26) => D26_INT
		EN --- MOVE(P10D27) => D27_INT
		EN --- MOVE(P10D28) => D28_INT
		EN --- MOVE(P10D29) => D29_INT
		EN --- MOVE(P10D30) => D30_INT
		EN --- MOVE(P10STG) => STG1_STG
NETWORK 47
	*
_END_LD_
(* the same logic as Structured Text *)
(* Network 1 *)
IF NOT LD_PB_IND_BOOL AND NPC THEN
	D00_INT := INT_D00;
	D01_INT := INT_D01;
	D02_INT := INT_D02;
	D03_INT := INT_D03;
	D04_INT := INT_D04;
	D05_INT := INT_D05;
	D06_INT := INT_D06;
	D07_INT := INT_D07;
	D08_INT := INT_D08;
	D09_INT := INT_D09;
	D10_INT := INT_D10;
	D11_INT := INT_D11;
	D12_INT := INT_D12;
	D13_INT := INT_D13;
	D14_INT := INT_D14;
	D15_INT := INT_D15;
	D16_INT := INT_D16;
	D17_INT := INT_D17;
	D18_INT := INT_D18;
	D19_INT := INT_D19;
	D20_INT := INT_D20;
	D21_INT := INT_D21;
	D22_INT := INT_D22;
	D23_INT := INT_D23;
	D24_INT := INT_D24;
	D25_INT := INT_D25;
	D26_INT := INT_D26;
	D27_INT := INT_D27;
	D28_INT := INT_D28;
	D29_INT := INT_D29;
	D30_INT := INT_D30;
	STG1_STG := STG_STG1;
END_IF;
(* Network 2 *)
P1B := INT_P_NO = 1;
(* Network 3 *)
P2B := INT_P_NO = 2;
(* Network 4 *)
P3B := INT_P_NO = 3;
(* Network 5 *)
P4B := INT_P_NO = 4;
(* Network 6 *)
P5B := INT_P_NO = 5;
(* Network 7 *)
P6B := INT_P_NO = 6;
(* Network 8 *)
P7B := INT_P_NO = 7;
(* Network 9 *)
P8B := INT_P_NO = 8;
(* Network 10 *)
P9B := INT_P_NO = 9;
(* Network 11 *)
P10B := INT_P_NO = 10;
(* Network 12 *)
TPC(IN := NOT N1, PT := T#300ms);
N0 := TPC.Q;
(* Network 13 *)
TPC1(IN := N0, PT := T#100ms);
N1 := TPC1.Q;
(* Network 14 *)
PCDF(CLK := N0);
PCTDF := PCDF.Q;
(* Network 15 *)
IF PCTDF THEN
	CNG_P_NO := INT_P_NO;
END_IF;
(* Network 16 *)
NPC := INT_P_NO = CNG_P_NO;
(* Network 17 *)
SVPLS(CLK := BOOL_SV_PB);
SV_PB_PLS := SVPLS.Q;
(* Network 18 *)
SV_HR := (SV_PB_PLS OR SV_HR) AND NOT SV_CR;
(* Network 19 *)
SV_T(IN := SV_HR, PT := T#1s);
SV_CR := SV_T.Q;
(* Network 20 *)
SV_PB_IND_BOOL := SV_HR;
(* Network 21 *)
SV_DF(CLK := SV_HR);
SV_PLS := SV_DF.Q;
(* Network 22 *)
IF SV_HR AND P1B THEN
	P01D00 := INT_D00;
	P01D01 := INT_D01;
	P01D02 := INT_D02;
	P01D03 := INT_D03;
	P01D04 := INT_D04;
	P01D05 := INT_D05;
	P01D06 := INT_D06;
	P01D07 := INT_D07;
	P01D08 := INT_D08;
	P01D09 := INT_D09;
	P01D10 := INT_D10;
	P01D11 := INT_D11;
	P01D12 := INT_D12;
	P01D13 := INT_D13;
	P01D14 := INT_D14;
	P01D15 := INT_D15;
	P01D16 := INT_D16;
	P01D17 := INT_D17;
	P01D18 := INT_D18;
	P01D19 := INT_D19;
	P01D20 := INT_D20;
	P01D21 := INT_D21;
	P01D22 := INT_D22;
	P01D23 := INT_D23;
	P01D24 := INT_D24;
	P01D25 := INT_D25;
	P01D26 := INT_D26;
	P01D27 := INT_D27;
	P01D28 := INT_D28;
	P01D29 := INT_D29;
	P01D30 := INT_D30;
	P01STG := STG_STG1;
END_IF;
(* Network 23 *)
IF SV_HR AND P2B THEN
	P02D00 := INT_D00;
	P02D01 := INT_D01;
	P02D02 := INT_D02;
	P02D03 := INT_D03;
	P02D04 := INT_D04;
	P02D05 := INT_D05;
	P02D06 := INT_D06;
	P02D07 := INT_D07;
	P02D08 := INT_D08;
	P02D09 := INT_D09;
	P02D10 := INT_D10;
	P02D11 := INT_D11;
	P02D12 := INT_D12;
	P02D13 := INT_D13;
	P02D14 := INT_D14;
	P02D15 := INT_D15;
	P02D16 := INT_D16;
	P02D17 := INT_D17;
	P02D18 := INT_D18;
	P02D19 := INT_D19;
	P02D20 := INT_D20;
	P02D21 := INT_D21;
	P02D22 := INT_D22;
	P02D23 := INT_D23;
	P02D24 := INT_D24;
	P02D25 := INT_D25;
	P02D26 := INT_D26;
	P02D27 := INT_D27;
	P02D28 := INT_D28;
	P02D29 := INT_D29;
	P02D30 := INT_D30;
	P02STG := STG_STG1;
END_IF;
(* Network 24 *)
IF SV_HR AND P3B THEN
	P03D00 := INT_D00;
	P03D01 := INT_D01;
	P03D02 := INT_D02;
	P03D03 := INT_D03;
	P03D04 := INT_D04;
	P03D05 := INT_D05;
	P03D06 := INT_D06;
	P03D07 := INT_D07;
	P03D08 := INT_D08;
	P03D09 := INT_D09;
	P03D10 := INT_D10;
	P03D11 := INT_D11;
	P03D12 := INT_D12;
	P03D13 := INT_D13;
	P03D14 := INT_D14;
	P03D15 := INT_D15;
	P03D16 := INT_D16;
	P03D17 := INT_D17;
	P03D18 := INT_D18;
	P03D19 := INT_D19;
	P03D20 := INT_D20;
	P03D21 := INT_D21;
	P03D22 := INT_D22;
	P03D23 := INT_D23;
	P03D24 := INT_D24;
	P03D25 := INT_D25;
	P03D26 := INT_D26;
	P03D27 := INT_D27;
	P03D28 := INT_D28;
	P03D29 := INT_D29;
	P03D30 := INT_D30;
	P03STG := STG_STG1;
END_IF;
(* Network 25 *)
IF SV_HR AND P4B THEN
	P04D00 := INT_D00;
	P04D01 := INT_D01;
	P04D02 := INT_D02;
	P04D03 := INT_D03;
	P04D04 := INT_D04;
	P04D05 := INT_D05;
	P04D06 := INT_D06;
	P04D07 := INT_D07;
	P04D08 := INT_D08;
	P04D09 := INT_D09;
	P04D10 := INT_D10;
	P04D11 := INT_D11;
	P04D12 := INT_D12;
	P04D13 := INT_D13;
	P04D14 := INT_D14;
	P04D15 := INT_D15;
	P04D16 := INT_D16;
	P04D17 := INT_D17;
	P04D18 := INT_D18;
	P04D19 := INT_D19;
	P04D20 := INT_D20;
	P04D21 := INT_D21;
	P04D22 := INT_D22;
	P04D23 := INT_D23;
	P04D24 := INT_D24;
	P04D25 := INT_D25;
	P04D26 := INT_D26;
	P04D27 := INT_D27;
	P04D28 := INT_D28;
	P04D29 := INT_D29;
	P04D30 := INT_D30;
	P04STG := STG_STG1;
END_IF;
(* Network 26 *)
IF SV_HR AND P5B THEN
	P05D00 := INT_D00;
	P05D01 := INT_D01;
	P05D02 := INT_D02;
	P05D03 := INT_D03;
	P05D04 := INT_D04;
	P05D05 := INT_D05;
	P05D06 := INT_D06;
	P05D07 := INT_D07;
	P05D08 := INT_D08;
	P05D09 := INT_D09;
	P05D10 := INT_D10;
	P05D11 := INT_D11;
	P05D12 := INT_D12;
	P05D13 := INT_D13;
	P05D14 := INT_D14;
	P05D15 := INT_D15;
	P05D16 := INT_D16;
	P05D17 := INT_D17;
	P05D18 := INT_D18;
	P05D19 := INT_D19;
	P05D20 := INT_D20;
	P05D21 := INT_D21;
	P05D22 := INT_D22;
	P05D23 := INT_D23;
	P05D24 := INT_D24;
	P05D25 := INT_D25;
	P05D26 := INT_D26;
	P05D27 := INT_D27;
	P05D28 := INT_D28;
	P05D29 := INT_D29;
	P05D30 := INT_D30;
	P05STG := STG_STG1;
END_IF;
(* Network 27 *)
IF SV_HR AND P6B THEN
	P06D00 := INT_D00;
	P06D01 := INT_D01;
	P06D02 := INT_D02;
	P06D03 := INT_D03;
	P06D04 := INT_D04;
	P06D05 := INT_D05;
	P06D06 := INT_D06;
	P06D07 := INT_D07;
	P06D08 := INT_D08;
	P06D09 := INT_D09;
	P06D10 := INT_D10;
	P06D11 := INT_D11;
	P06D12 := INT_D12;
	P06D13 := INT_D13;
	P06D14 := INT_D14;
	P06D15 := INT_D15;
	P06D16 := INT_D16;
	P06D17 := INT_D17;
	P06D18 := INT_D18;
	P06D19 := INT_D19;
	P06D20 := INT_D20;
	P06D21 := INT_D21;
	P06D22 := INT_D22;
	P06D23 := INT_D23;
	P06D24 := INT_D24;
	P06D25 := INT_D25;
	P06D26 := INT_D26;
	P06D27 := INT_D27;
	P06D28 := INT_D28;
	P06D29 := INT_D29;
	P06D30 := INT_D30;
	P06STG := STG_STG1;
END_IF;
(* Network 28 *)
IF SV_HR AND P7B THEN
	P07D00 := INT_D00;
	P07D01 := INT_D01;
	P07D02 := INT_D02;
	P07D03 := INT_D03;
	P07D04 := INT_D04;
	P07D05 := INT_D05;
	P07D06 := INT_D06;
	P07D07 := INT_D07;
	P07D08 := INT_D08;
	P07D09 := INT_D09;
	P07D10 := INT_D10;
	P07D11 := INT_D11;
	P07D12 := INT_D12;
	P07D13 := INT_D13;
	P07D14 := INT_D14;
	P07D15 := INT_D15;
	P07D16 := INT_D16;
	P07D17 := INT_D17;
	P07D18 := INT_D18;
	P07D19 := INT_D19;
	P07D20 := INT_D20;
	P07D21 := INT_D21;
	P07D22 := INT_D22;
	P07D23 := INT_D23;
	P07D24 := INT_D24;
	P07D25 := INT_D25;
	P07D26 := INT_D26;
	P07D27 := INT_D27;
	P07D28 := INT_D28;
	P07D29 := INT_D29;
	P07D30 := INT_D30;
	P07STG := STG_STG1;
END_IF;
(* Network 29 *)
IF SV_HR AND P8B THEN
	P08D00 := INT_D00;
	P08D01 := INT_D01;
	P08D02 := INT_D02;
	P08D03 := INT_D03;
	P08D04 := INT_D04;
	P08D05 := INT_D05;
	P08D06 := INT_D06;
	P08D07 := INT_D07;
	P08D08 := INT_D08;
	P08D09 := INT_D09;
	P08D10 := INT_D10;
	P08D11 := INT_D11;
	P08D12 := INT_D12;
	P08D13 := INT_D13;
	P08D14 := INT_D14;
	P08D15 := INT_D15;
	P08D16 := INT_D16;
	P08D17 := INT_D17;
	P08D18 := INT_D18;
	P08D19 := INT_D19;
	P08D20 := INT_D20;
	P08D21 := INT_D21;
	P08D22 := INT_D22;
	P08D23 := INT_D23;
	P08D24 := INT_D24;
	P08D25 := INT_D25;
	P08D26 := INT_D26;
	P08D27 := INT_D27;
	P08D28 := INT_D28;
	P08D29 := INT_D29;
	P08D30 := INT_D30;
	P08STG := STG_STG1;
END_IF;
(* Network 30 *)
IF SV_HR AND P9B THEN
	P09D00 := INT_D00;
	P09D01 := INT_D01;
	P09D02 := INT_D02;
	P09D03 := INT_D03;
	P09D04 := INT_D04;
	P09D05 := INT_D05;
	P09D06 := INT_D06;
	P09D07 := INT_D07;
	P09D08 := INT_D08;
	P09D09 := INT_D09;
	P09D10 := INT_D10;
	P09D11 := INT_D11;
	P09D12 := INT_D12;
	P09D13 := INT_D13;
	P09D14 := INT_D14;
	P09D15 := INT_D15;
	P09D16 := INT_D16;
	P09D17 := INT_D17;
	P09D18 := INT_D18;
	P09D19 := INT_D19;
	P09D20 := INT_D20;
	P09D21 := INT_D21;
	P09D22 := INT_D22;
	P09D23 := INT_D23;
	P09D24 := INT_D24;
	P09D25 := INT_D25;
	P09D26 := INT_D26;
	P09D27 := INT_D27;
	P09D28 := INT_D28;
	P09D29 := INT_D29;
	P09D30 := INT_D30;
	P09STG := STG_STG1;
END_IF;
(* Network 31 *)
IF SV_HR AND P10B THEN
	P10D00 := INT_D00;
	P10D01 := INT_D01;
	P10D02 := INT_D02;
	P10D03 := INT_D03;
	P10D04 := INT_D04;
	P10D05 := INT_D05;
	P10D06 := INT_D06;
	P10D07 := INT_D07;
	P10D08 := INT_D08;
	P10D09 := INT_D09;
	P10D10 := INT_D10;
	P10D11 := INT_D11;
	P10D12 := INT_D12;
	P10D13 := INT_D13;
	P10D14 := INT_D14;
	P10D15 := INT_D15;
	P10D16 := INT_D16;
	P10D17 := INT_D17;
	P10D18 := INT_D18;
	P10D19 := INT_D19;
	P10D20 := INT_D20;
	P10D21 := INT_D21;
	P10D22 := INT_D22;
	P10D23 := INT_D23;
	P10D24 := INT_D24;
	P10D25 := INT_D25;
	P10D26 := INT_D26;
	P10D27 := INT_D27;
	P10D28 := INT_D28;
	P10D29 := INT_D29;
	P10D30 := INT_D30;
	P10STG := STG_STG1;
END_IF;
(* Network 32 *)
LDPLS(CLK := BOOL_LD_PB);
LD_PB_PLS := LDPLS.Q;
(* Network 33 *)
LD_HR := (LD_PB_PLS OR LD_HR) AND NOT LD_CR;
(* Network 34 *)
LD_T(IN := LD_HR, PT := T#1s);
LD_CR := LD_T.Q;
(* Network 35 *)
LD_PB_IND_BOOL := LD_HR;
(* Network 36 *)
LD_DF(CLK := LD_HR);
LD_PLS := LD_DF.Q;
(* Network 37 *)
IF (LD_HR OR NOT NPC) AND P1B THEN
	D00_INT := P01D00;
	D01_INT := P01D01;
	D02_INT := P01D02;
	D03_INT := P01D03;
	D04_INT := P01D04;
	D05_INT := P01D05;
	D06_INT := P01D06;
	D07_INT := P01D07;
	D08_INT := P01D08;
	D09_INT := P01D09;
	D10_INT := P01D10;
	D11_INT := P01D11;
	D12_INT := P01D12;
	D13_INT := P01D13;
	D14_INT := P01D14;
	D15_INT := P01D15;
	D16_INT := P01D16;
	D17_INT := P01D17;
	D18_INT := P01D18;
	D19_INT := P01D19;
	D20_INT := P01D20;
	D21_INT := P01D21;
	D22_INT := P01D22;
	D23_INT := P01D23;
	D24_INT := P01D24;
	D25_INT := P01D25;
	D26_INT := P01D26;
	D27_INT := P01D27;
	D28_INT := P01D28;
	D29_INT := P01D29;
	D30_INT := P01D30;
	STG1_STG := P01STG;
END_IF;
(* Network 38 *)
IF (LD_HR OR NOT NPC) AND P2B THEN
	D00_INT := P02D00;
	D01_INT := P02D01;
	D02_INT := P02D02;
	D03_INT := P02D03;
	D04_INT := P02D04;
	D05_INT := P02D05;
	D06_INT := P02D06;
	D07_INT := P02D07;
	D08_INT := P02D08;
	D09_INT := P02D09;
	D10_INT := P02D10;
	D11_INT := P02D11;
	D12_INT := P02D12;
	D13_INT := P02D13;
	D14_INT := P02D14;
	D15_INT := P02D15;
	D16_INT := P02D16;
	D17_INT := P02D17;
	D18_INT := P02D18;
	D19_INT := P02D19;
	D20_INT := P02D20;
	D21_INT := P02D21;
	D22_INT := P02D22;
	D23_INT := P02D23;
	D24_INT := P02D24;
	D25_INT := P02D25;
	D26_INT := P02D26;
	D27_INT := P02D27;
	D28_INT := P02D28;
	D29_INT := P02D29;
	D30_INT := P02D30;
	STG1_STG := P02STG;
END_IF;
(* Network 39 *)
IF (LD_HR OR NOT NPC) AND P3B THEN
	D00_INT := P03D00;
	D01_INT := P03D01;
	D02_INT := P03D02;
	D03_INT := P03D03;
	D04_INT := P03D04;
	D05_INT := P03D05;
	D06_INT := P03D06;
	D07_INT := P03D07;
	D08_INT := P03D08;
	D09_INT := P03D09;
	D10_INT := P03D10;
	D11_INT := P03D11;
	D12_INT := P03D12;
	D13_INT := P03D13;
	D14_INT := P03D14;
	D15_INT := P03D15;
	D16_INT := P03D16;
	D17_INT := P03D17;
	D18_INT := P03D18;
	D19_INT := P03D19;
	D20_INT := P03D20;
	D21_INT := P03D21;
	D22_INT := P03D22;
	D23_INT := P03D23;
	D24_INT := P03D24;
	D25_INT := P03D25;
	D26_INT := P03D26;
	D27_INT := P03D27;
	D28_INT := P03D28;
	D29_INT := P03D29;
	D30_INT := P03D30;
	STG1_STG := P03STG;
END_IF;
(* Network 40 *)
IF (LD_HR OR NOT NPC) AND P4B THEN
	D00_INT := P04D00;
	D01_INT := P04D01;
	D02_INT := P04D02;
	D03_INT := P04D03;
	D04_INT := P04D04;
	D05_INT := P04D05;
	D06_INT := P04D06;
	D07_INT := P04D07;
	D08_INT := P04D08;
	D09_INT := P04D09;
	D10_INT := P04D10;
	D11_INT := P04D11;
	D12_INT := P04D12;
	D13_INT := P04D13;
	D14_INT := P04D14;
	D15_INT := P04D15;
	D16_INT := P04D16;
	D17_INT := P04D17;
	D18_INT := P04D18;
	D19_INT := P04D19;
	D20_INT := P04D20;
	D21_INT := P04D21;
	D22_INT := P04D22;
	D23_INT := P04D23;
	D24_INT := P04D24;
	D25_INT := P04D25;
	D26_INT := P04D26;
	D27_INT := P04D27;
	D28_INT := P04D28;
	D29_INT := P04D29;
	D30_INT := P04D30;
	STG1_STG := P04STG;
END_IF;
(* Network 41 *)
IF (LD_HR OR NOT NPC) AND P5B THEN
	D00_INT := P05D00;
	D01_INT := P05D01;
	D02_INT := P05D02;
	D03_INT := P05D03;
	D04_INT := P05D04;
	D05_INT := P05D05;
	D06_INT := P05D06;
	D07_INT := P05D07;
	D08_INT := P05D08;
	D09_INT := P05D09;
	D10_INT := P05D10;
	D11_INT := P05D11;
	D12_INT := P05D12;
	D13_INT := P05D13;
	D14_INT := P05D14;
	D15_INT := P05D15;
	D16_INT := P05D16;
	D17_INT := P05D17;
	D18_INT := P05D18;
	D19_INT := P05D19;
	D20_INT := P05D20;
	D21_INT := P05D21;
	D22_INT := P05D22;
	D23_INT := P05D23;
	D24_INT := P05D24;
	D25_INT := P05D25;
	D26_INT := P05D26;
	D27_INT := P05D27;
	D28_INT := P05D28;
	D29_INT := P05D29;
	D30_INT := P05D30;
	STG1_STG := P05STG;
END_IF;
(* Network 42 *)
IF (LD_HR OR NOT NPC) AND P6B THEN
	D00_INT := P06D00;
	D01_INT := P06D01;
	D02_INT := P06D02;
	D03_INT := P06D03;
	D04_INT := P06D04;
	D05_INT := P06D05;
	D06_INT := P06D06;
	D07_INT := P06D07;
	D08_INT := P06D08;
	D09_INT := P06D09;
	D10_INT := P06D10;
	D11_INT := P06D11;
	D12_INT := P06D12;
	D13_INT := P06D13;
	D14_INT := P06D14;
	D15_INT := P06D15;
	D16_INT := P06D16;
	D17_INT := P06D17;
	D18_INT := P06D18;
	D19_INT := P06D19;
	D20_INT := P06D20;
	D21_INT := P06D21;
	D22_INT := P06D22;
	D23_INT := P06D23;
	D24_INT := P06D24;
	D25_INT := P06D25;
	D26_INT := P06D26;
	D27_INT := P06D27;
	D28_INT := P06D28;
	D29_INT := P06D29;
	D30_INT := P06D30;
	STG1_STG := P06STG;
END_IF;
(* Network 43 *)
IF (LD_HR OR NOT NPC) AND P7B THEN
	D00_INT := P07D00;
	D01_INT := P07D01;
	D02_INT := P07D02;
	D03_INT := P07D03;
	D04_INT := P07D04;
	D05_INT := P07D05;
	D06_INT := P07D06;
	D07_INT := P07D07;
	D08_INT := P07D08;
	D09_INT := P07D09;
	D10_INT := P07D10;
	D11_INT := P07D11;
	D12_INT := P07D12;
	D13_INT := P07D13;
	D14_INT := P07D14;
	D15_INT := P07D15;
	D16_INT := P07D16;
	D17_INT := P07D17;
	D18_INT := P07D18;
	D19_INT := P07D19;
	D20_INT := P07D20;
	D21_INT := P07D21;
	D22_INT := P07D22;
	D23_INT := P07D23;
	D24_INT := P07D24;
	D25_INT := P07D25;
	D26_INT := P07D26;
	D27_INT := P07D27;
	D28_INT := P07D28;
	D29_INT := P07D29;
	D30_INT := P07D30;
	STG1_STG := P07STG;
END_IF;
(* Network 44 *)
IF (LD_HR OR NOT NPC) AND P8B THEN
	D00_INT := P08D00;
	D01_INT := P08D01;
	D02_INT := P08D02;
	D03_INT := P08D03;
	D04_INT := P08D04;
	D05_INT := P08D05;
	D06_INT := P08D06;
	D07_INT := P08D07;
	D08_INT := P08D08;
	D09_INT := P08D09;
	D10_INT := P08D10;
	D11_INT := P08D11;
	D12_INT := P08D12;
	D13_INT := P08D13;
	D14_INT := P08D14;
	D15_INT := P08D15;
	D16_INT := P08D16;
	D17_INT := P08D17;
	D18_INT := P08D18;
	D19_INT := P08D19;
	D20_INT := P08D20;
	D21_INT := P08D21;
	D22_INT := P08D22;
	D23_INT := P08D23;
	D24_INT := P08D24;
	D25_INT := P08D25;
	D26_INT := P08D26;
	D27_INT := P08D27;
	D28_INT := P08D28;
	D29_INT := P08D29;
	D30_INT := P08D30;
	STG1_STG := P08STG;
END_IF;
(* Network 45 *)
IF (LD_HR OR NOT NPC) AND P9B THEN
	D00_INT := P09D00;
	D01_INT := P09D01;
	D02_INT := P09D02;
	D03_INT := P09D03;
	D04_INT := P09D04;
	D05_INT := P09D05;
	D06_INT := P09D06;
	D07_INT := P09D07;
	D08_INT := P09D08;
	D09_INT := P09D09;
	D10_INT := P09D10;
	D11_INT := P09D11;
	D12_INT := P09D12;
	D13_INT := P09D13;
	D14_INT := P09D14;
	D15_INT := P09D15;
	D16_INT := P09D16;
	D17_INT := P09D17;
	D18_INT := P09D18;
	D19_INT := P09D19;
	D20_INT := P09D20;
	D21_INT := P09D21;
	D22_INT := P09D22;
	D23_INT := P09D23;
	D24_INT := P09D24;
	D25_INT := P09D25;
	D26_INT := P09D26;
	D27_INT := P09D27;
	D28_INT := P09D28;
	D29_INT := P09D29;
	D30_INT := P09D30;
	STG1_STG := P09STG;
END_IF;
(* Network 46 *)
IF (LD_HR OR NOT NPC) AND P10B THEN
	D00_INT := P10D00;
	D01_INT := P10D01;
	D02_INT := P10D02;
	D03_INT := P10D03;
	D04_INT := P10D04;
	D05_INT := P10D05;
	D06_INT := P10D06;
	D07_INT := P10D07;
	D08_INT := P10D08;
	D09_INT := P10D09;
	D10_INT := P10D10;
	D11_INT := P10D11;
	D12_INT := P10D12;
	D13_INT := P10D13;
	D14_INT := P10D14;
	D15_INT := P10D15;
	D16_INT := P10D16;
	D17_INT := P10D17;
	D18_INT := P10D18;
	D19_INT := P10D19;
	D20_INT := P10D20;
	D21_INT := P10D21;
	D22_INT := P10D22;
	D23_INT := P10D23;
	D24_INT := P10D24;
	D25_INT := P10D25;
	D26_INT := P10D26;
	D27_INT := P10D27;
	D28_INT := P10D28;
	D29_INT := P10D29;
	D30_INT := P10D30;
	STG1_STG := P10STG;
END_IF;
(* Network 47 *)
END_FUNCTION_BLOCK

(* POU JOG_CONV, LD *)
FUNCTION_BLOCK JOG_CONV
VAR_INPUT
	BOOL_FWD_JOG : BOOL;
	BOOL_RWD_JOG : BOOL;
	UINT_JOG_SPD_MM : UINT;
	TIME_JOG_DELAY : TIME;
	UINT_PLS_RATIO : UINT;

END_VAR
VAR_OUTPUT
	JOG_ACTIVE_BOOL : BOOL;
	JOG_SPD_UINT : UINT;


END_VAR
VAR
	VUINT: UINT;
	T1: TON;
	TI: TIME;
	JSPD_PLS: UINT;
END_VAR
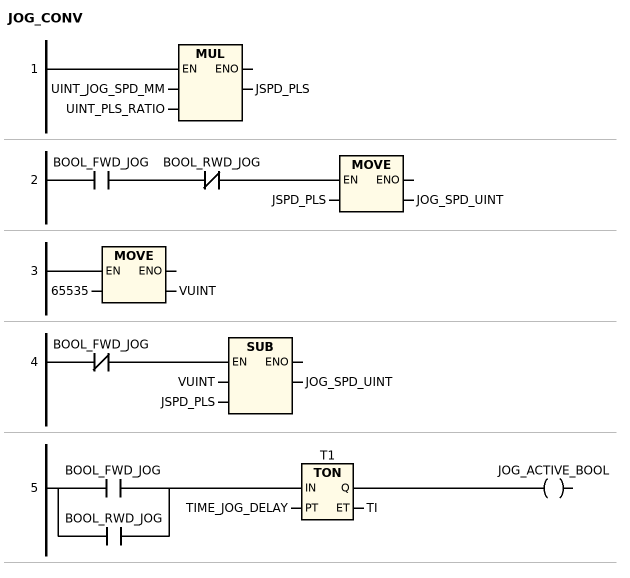
_LD_ (* Ladder Diagram *)
NETWORK 1
	*
		EN --- MUL(UINT_JOG_SPD_MM, UINT_PLS_RATIO) => JSPD_PLS
NETWORK 2
	[BOOL_FWD_JOG] - [/BOOL_RWD_JOG]
		EN --- MOVE(JSPD_PLS) => JOG_SPD_UINT
NETWORK 3
	*
		EN --- MOVE(65535) => VUINT
NETWORK 4
	[/BOOL_FWD_JOG]
		EN --- SUB(VUINT, JSPD_PLS) => JOG_SPD_UINT
NETWORK 5
	{ [BOOL_FWD_JOG] | [BOOL_RWD_JOG] } - T1:TON(IN: *, PT: TIME_JOG_DELAY, ET => TI) --- (JOG_ACTIVE_BOOL)
_END_LD_
(* the same logic as Structured Text *)
(* Network 1 *)
JSPD_PLS := UINT_JOG_SPD_MM * UINT_PLS_RATIO;
(* Network 2 *)
IF BOOL_FWD_JOG AND NOT BOOL_RWD_JOG THEN
	JOG_SPD_UINT := JSPD_PLS;
END_IF;
(* Network 3 *)
VUINT := 65535;
(* Network 4 *)
IF NOT BOOL_FWD_JOG THEN
	JOG_SPD_UINT := VUINT - JSPD_PLS;
END_IF;
(* Network 5 *)
T1(IN := BOOL_FWD_JOG OR BOOL_RWD_JOG, PT := TIME_JOG_DELAY);
TI := T1.ET;
JOG_ACTIVE_BOOL := T1.Q;
END_FUNCTION_BLOCK

(* POU LT_GT, LD *)
FUNCTION_BLOCK LT_GT
VAR_INPUT
	INT_SOURCE_A: INT;
	INT_SOURCE_B: INT;
END_VAR
VAR_OUTPUT
	SIGNAL_BOOL: BOOL;
END_VAR
VAR
	M0: BOOL;
	M1: BOOL;
END_VAR
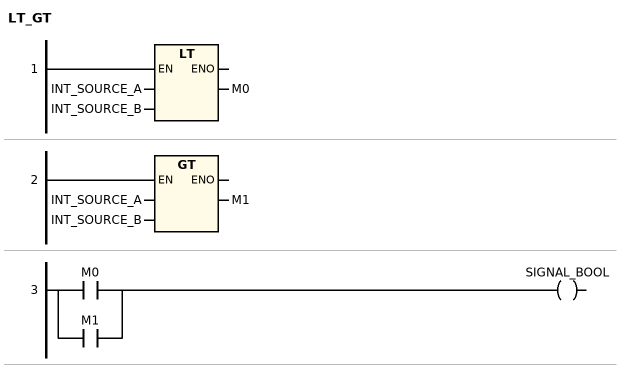
_LD_ (* Ladder Diagram *)
NETWORK 1
	*
		EN --- LT(INT_SOURCE_A, INT_SOURCE_B) => M0
NETWORK 2
	*
		EN --- GT(INT_SOURCE_A, INT_SOURCE_B) => M1
NETWORK 3
	{ [M0] | [M1] } --- (SIGNAL_BOOL)
_END_LD_
(* the same logic as Structured Text *)
(* Network 1 *)
M0 := INT_SOURCE_A < INT_SOURCE_B;
(* Network 2 *)
M1 := INT_SOURCE_A > INT_SOURCE_B;
(* Network 3 *)
SIGNAL_BOOL := M0 OR M1;
END_FUNCTION_BLOCK

(* POU MANUAL_PAGE, FBD *)
FUNCTION_BLOCK MANUAL_PAGE
VAR_INPUT
	STRING_PG1 : STRING;
	STRING_PG2 : STRING;
	STRING_PG3 : STRING;
	STRING_PG4 : STRING;
	STRING_PG5 : STRING;
	STRING_PG6 : STRING;
	STRING_PG7 : STRING;
	STRING_PG8 : STRING;
	STRING_PG9 : STRING;
	STRING_PG10 : STRING;
	STRING_PG11 : STRING;
	STRING_PG12 : STRING;
	STRING_PG13 : STRING;
	STRING_PG14 : STRING;
	STRING_PG15 : STRING;
	STRING_PG16 : STRING;
	STRING_PG17 : STRING;
	STRING_PG18 : STRING;
	STRING_PG19 : STRING;
	STRING_PG20 : STRING;
	STRING_CVISU : STRING;


END_VAR
VAR_OUTPUT
	PG_CONFIRMED_BOOL : BOOL;

END_VAR
VAR
END_VAR
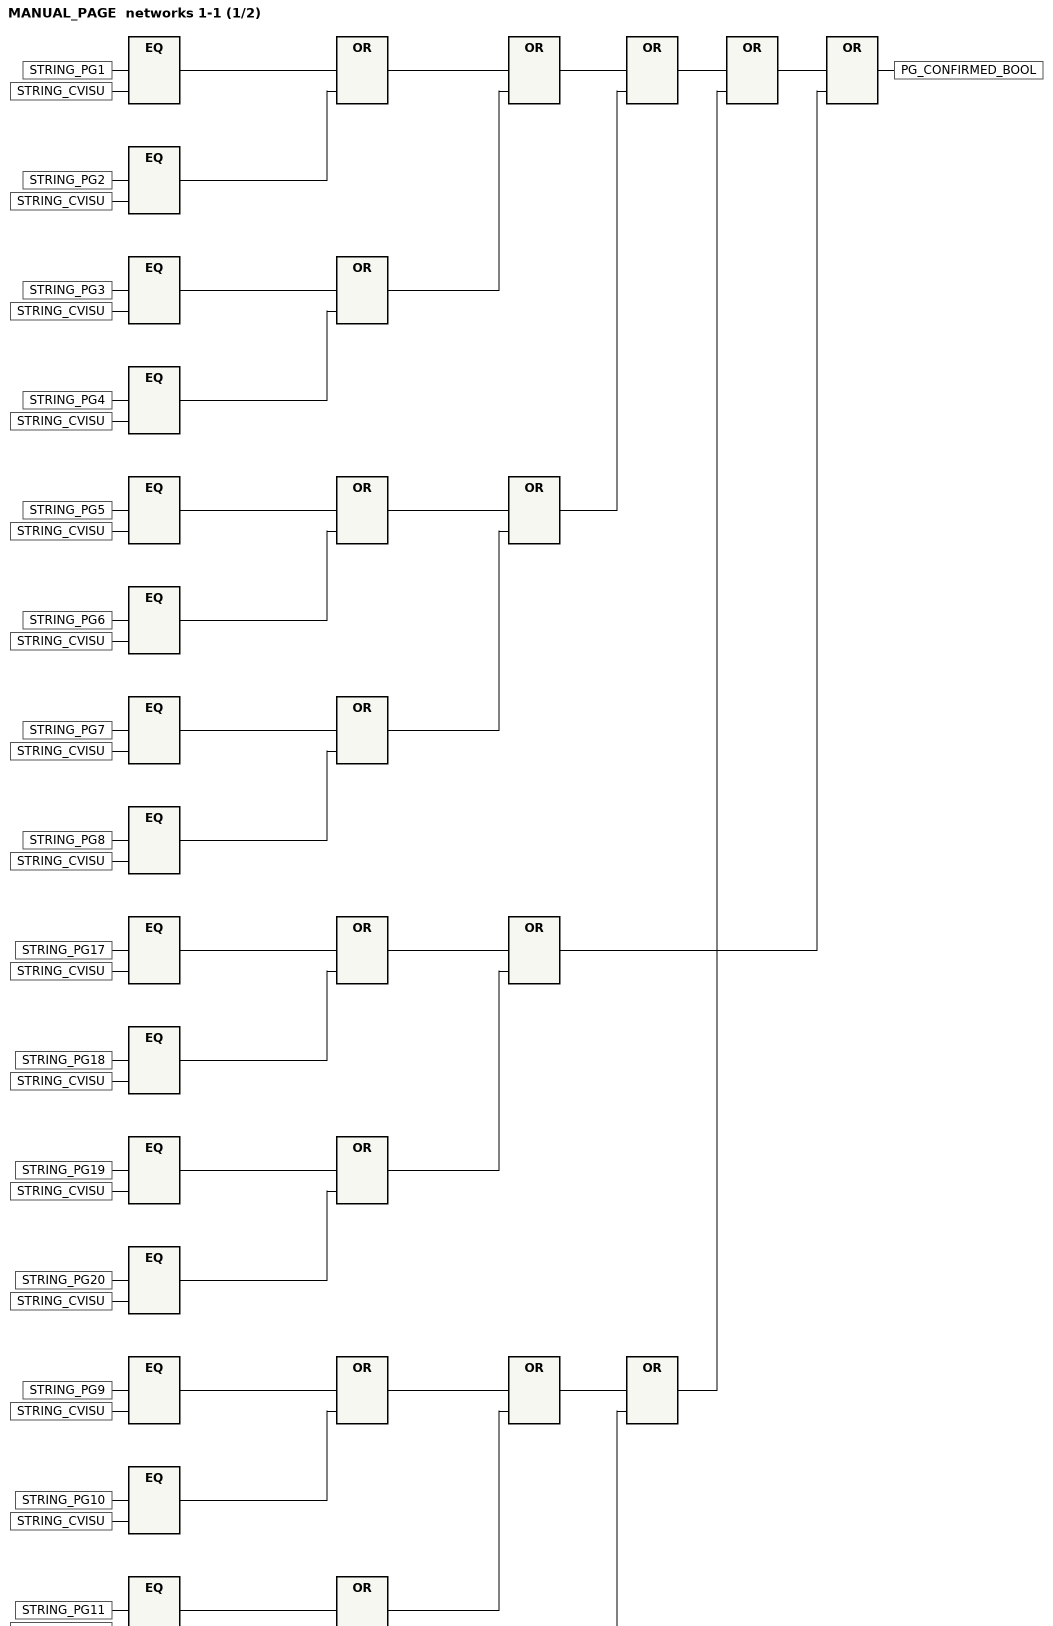
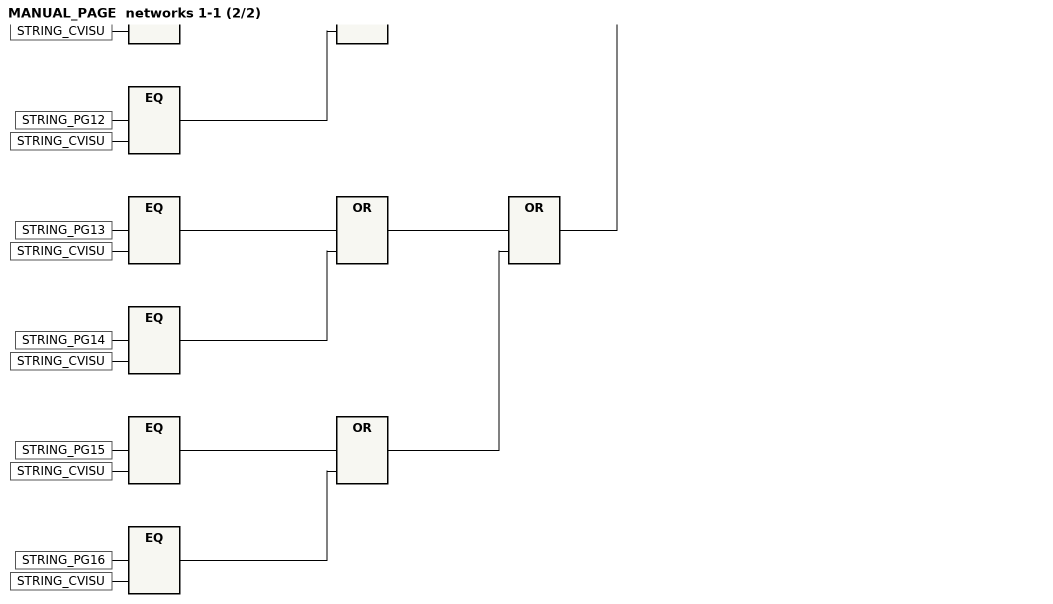
_FBD_ (* Function Block Diagram *)
NETWORK 1
	OR(OR(OR(OR(OR(EQ(STRING_PG1, STRING_CVISU), EQ(STRING_PG2, STRING_CVISU)), OR(EQ(STRING_PG3, STRING_CVISU), EQ(STRING_PG4, STRING_CVISU))), OR(OR(EQ(STRING_PG5, STRING_CVISU), EQ(STRING_PG6, STRING_CVISU)), OR(EQ(STRING_PG7, STRING_CVISU), EQ(STRING_PG8, STRING_CVISU)))), OR(OR(OR(EQ(STRING_PG9, STRING_CVISU), EQ(STRING_PG10, STRING_CVISU)), OR(EQ(STRING_PG11, STRING_CVISU), EQ(STRING_PG12, STRING_CVISU))), OR(OR(EQ(STRING_PG13, STRING_CVISU), EQ(STRING_PG14, STRING_CVISU)), OR(EQ(STRING_PG15, STRING_CVISU), EQ(STRING_PG16, STRING_CVISU))))), OR(OR(EQ(STRING_PG17, STRING_CVISU), EQ(STRING_PG18, STRING_CVISU)), OR(EQ(STRING_PG19, STRING_CVISU), EQ(STRING_PG20, STRING_CVISU)))) => PG_CONFIRMED_BOOL
_END_FBD_
(* the same logic as Structured Text *)
(* Network 1 *)
PG_CONFIRMED_BOOL := (((((STRING_PG1 = STRING_CVISU) OR (STRING_PG2 = STRING_CVISU)) OR ((STRING_PG3 = STRING_CVISU) OR (STRING_PG4 = STRING_CVISU))) OR (((STRING_PG5 = STRING_CVISU) OR (STRING_PG6 = STRING_CVISU)) OR ((STRING_PG7 = STRING_CVISU) OR (STRING_PG8 = STRING_CVISU)))) OR ((((STRING_PG9 = STRING_CVISU) OR (STRING_PG10 = STRING_CVISU)) OR ((STRING_PG11 = STRING_CVISU) OR (STRING_PG12 = STRING_CVISU))) OR (((STRING_PG13 = STRING_CVISU) OR (STRING_PG14 = STRING_CVISU)) OR ((STRING_PG15 = STRING_CVISU) OR (STRING_PG16 = STRING_CVISU))))) OR (((STRING_PG17 = STRING_CVISU) OR (STRING_PG18 = STRING_CVISU)) OR ((STRING_PG19 = STRING_CVISU) OR (STRING_PG20 = STRING_CVISU)));
END_FUNCTION_BLOCK

(* POU MM_TO_PLS, FBD *)
FUNCTION_BLOCK MM_TO_PLS
VAR_INPUT
	UINT_PLS_RATIO : UINT;
	UINT_TARGET1_MM : UINT;
	UINT_VEL1_MM : UINT;
	UINT_TARGET2_MM : UINT;
	UINT_VEL2_MM : UINT;
	UINT_TARGET3_MM : UINT;
	UINT_VEL3_MM : UINT;
	UINT_TARGET4_MM : UINT;
	UINT_VEL4_MM : UINT;
	UINT_JOG_2SPD_MM : UINT;
END_VAR

VAR_OUTPUT
	TARGET1_WR_UINT : UINT;
	VEL1_WR_UINT : UINT;
	TARGET2_WR_UINT : UINT;
	VEL2_WR_UINT : UINT;
	TARGET3_WR_UINT : UINT;
	VEL3_WR_UINT : UINT;
	TARGET4_WR_UINT : UINT;
	VEL4_WR_UINT : UINT;
	JOG_2SPD_UINT : UINT;

END_VAR

VAR
END_VAR
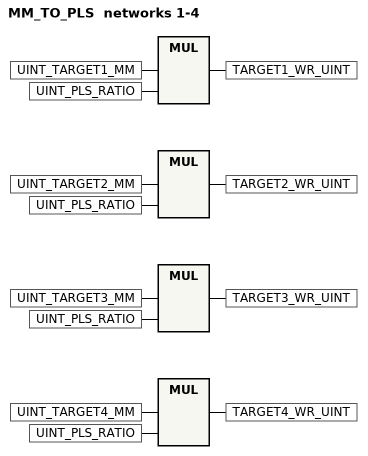
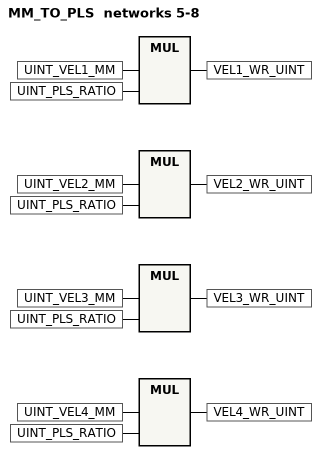
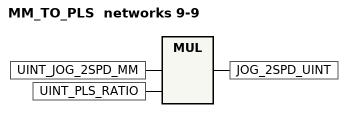
_FBD_ (* Function Block Diagram *)
NETWORK 1
	MUL(UINT_TARGET1_MM, UINT_PLS_RATIO) => TARGET1_WR_UINT
NETWORK 2
	MUL(UINT_TARGET2_MM, UINT_PLS_RATIO) => TARGET2_WR_UINT
NETWORK 3
	MUL(UINT_TARGET3_MM, UINT_PLS_RATIO) => TARGET3_WR_UINT
NETWORK 4
	MUL(UINT_TARGET4_MM, UINT_PLS_RATIO) => TARGET4_WR_UINT
NETWORK 5
	MUL(UINT_VEL1_MM, UINT_PLS_RATIO) => VEL1_WR_UINT
NETWORK 6
	MUL(UINT_VEL2_MM, UINT_PLS_RATIO) => VEL2_WR_UINT
NETWORK 7
	MUL(UINT_VEL3_MM, UINT_PLS_RATIO) => VEL3_WR_UINT
NETWORK 8
	MUL(UINT_VEL4_MM, UINT_PLS_RATIO) => VEL4_WR_UINT
NETWORK 9
	MUL(UINT_JOG_2SPD_MM, UINT_PLS_RATIO) => JOG_2SPD_UINT
_END_FBD_
(* the same logic as Structured Text *)
(* Network 1 *)
TARGET1_WR_UINT := UINT_TARGET1_MM * UINT_PLS_RATIO;
(* Network 2 *)
TARGET2_WR_UINT := UINT_TARGET2_MM * UINT_PLS_RATIO;
(* Network 3 *)
TARGET3_WR_UINT := UINT_TARGET3_MM * UINT_PLS_RATIO;
(* Network 4 *)
TARGET4_WR_UINT := UINT_TARGET4_MM * UINT_PLS_RATIO;
(* Network 5 *)
VEL1_WR_UINT := UINT_VEL1_MM * UINT_PLS_RATIO;
(* Network 6 *)
VEL2_WR_UINT := UINT_VEL2_MM * UINT_PLS_RATIO;
(* Network 7 *)
VEL3_WR_UINT := UINT_VEL3_MM * UINT_PLS_RATIO;
(* Network 8 *)
VEL4_WR_UINT := UINT_VEL4_MM * UINT_PLS_RATIO;
(* Network 9 *)
JOG_2SPD_UINT := UINT_JOG_2SPD_MM * UINT_PLS_RATIO;
END_FUNCTION_BLOCK

(* POU MOTION_ACC_DCC, LD *)
FUNCTION_BLOCK MOTION_ACC_DCC
VAR_INPUT
	BOOL_UP_MOVE : BOOL;
	BOOL_DOWN_MOVE : BOOL;
	UINT_JOG_ACCDCC : UINT;
	UINT_HOME_ACCDCC : UINT;
	UINT_UD_ACCDCC : UINT;
	UINT_AG_ACCDCC : UINT;
	TIME_UD_DLY_ON : TIME;
	BOOL_MANUAL_PG : BOOL;
	BOOL_ORIGIN_COMP : BOOL;
	BOOL_ARM_HOME_READY : BOOL;
	STRING_CURRENT_PG : STRING;
	STRING_MAN_JOG_V_PG : STRING;
	STRING_MAN_POS_V_PG : STRING;
	STRING_MAN_JOG_H_PG : STRING;
	STRING_MAN_POS_H_PG : STRING;
END_VAR
VAR_OUTPUT

	UP_MOVE_ST_BOOL : BOOL;
	DOWN_MOVE_ST_BOOL : BOOL;
	ACC_UINT : UINT;
	DCC_UINT : UINT;

END_VAR
VAR
	T1: TON;
	T1COUNT: TIME;
	T2: TON;
	T2COUNT: TIME;
	MANJOGH: BOOL;
	MANJOGV: BOOL;
	MANPOSH: BOOL;
	MANPOSV: BOOL;
END_VAR
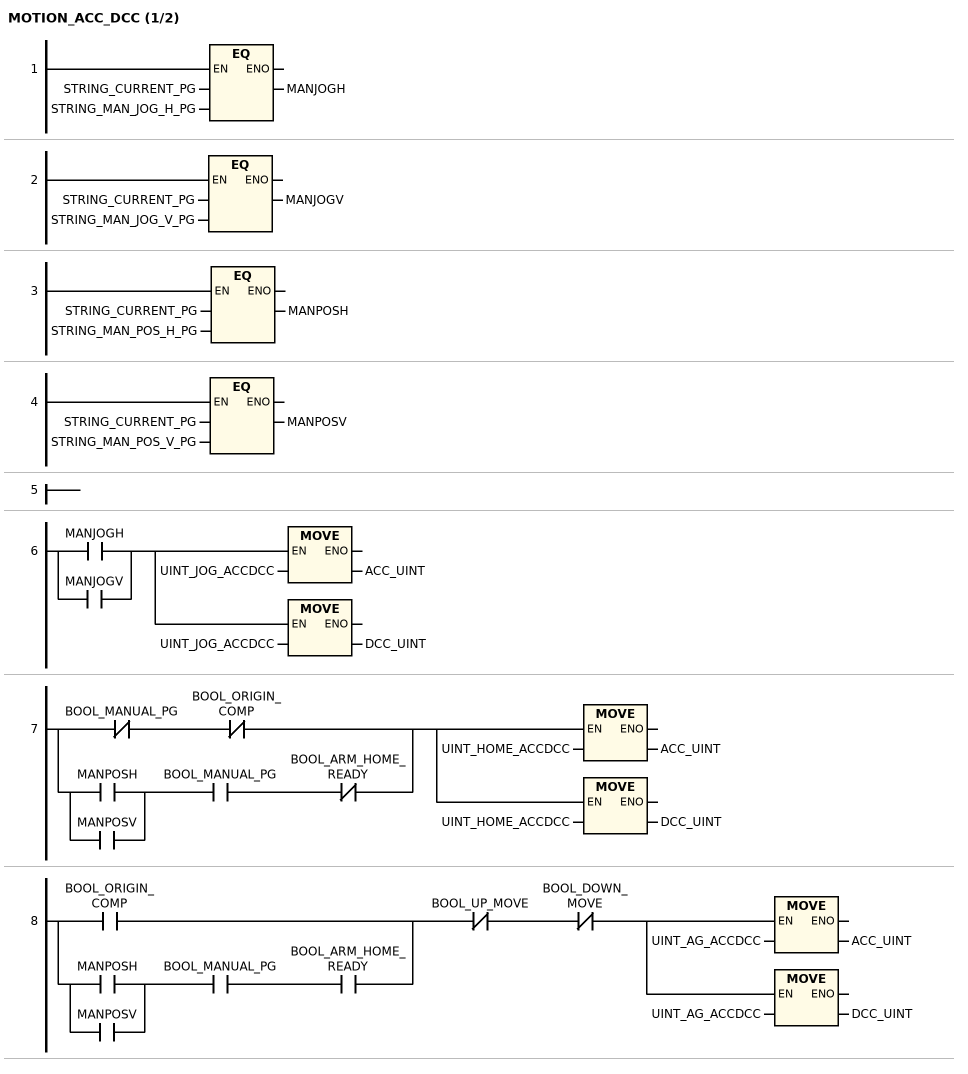
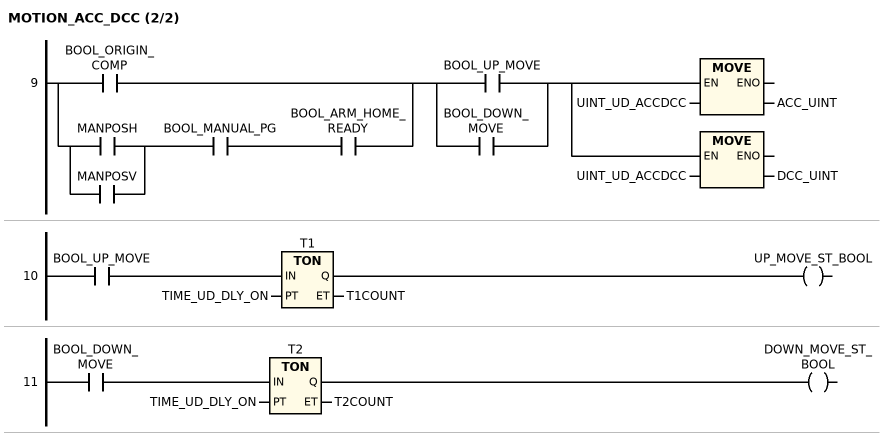
_LD_ (* Ladder Diagram *)
NETWORK 1
	*
		EN --- EQ(STRING_CURRENT_PG, STRING_MAN_JOG_H_PG) => MANJOGH
NETWORK 2
	*
		EN --- EQ(STRING_CURRENT_PG, STRING_MAN_JOG_V_PG) => MANJOGV
NETWORK 3
	*
		EN --- EQ(STRING_CURRENT_PG, STRING_MAN_POS_H_PG) => MANPOSH
NETWORK 4
	*
		EN --- EQ(STRING_CURRENT_PG, STRING_MAN_POS_V_PG) => MANPOSV
NETWORK 5
	*
NETWORK 6
	{ [MANJOGH] | [MANJOGV] }
		EN --- MOVE(UINT_JOG_ACCDCC) => ACC_UINT
		EN --- MOVE(UINT_JOG_ACCDCC) => DCC_UINT
NETWORK 7
	{ [/BOOL_MANUAL_PG] - [/BOOL_ORIGIN_COMP] | { [MANPOSH] | [MANPOSV] } - [BOOL_MANUAL_PG] - [/BOOL_ARM_HOME_READY] }
		EN --- MOVE(UINT_HOME_ACCDCC) => ACC_UINT
		EN --- MOVE(UINT_HOME_ACCDCC) => DCC_UINT
NETWORK 8
	{ [BOOL_ORIGIN_COMP] | { [MANPOSH] | [MANPOSV] } - [BOOL_MANUAL_PG] - [BOOL_ARM_HOME_READY] } - [/BOOL_UP_MOVE] - [/BOOL_DOWN_MOVE]
		EN --- MOVE(UINT_AG_ACCDCC) => ACC_UINT
		EN --- MOVE(UINT_AG_ACCDCC) => DCC_UINT
NETWORK 9
	{ [BOOL_ORIGIN_COMP] | { [MANPOSH] | [MANPOSV] } - [BOOL_MANUAL_PG] - [BOOL_ARM_HOME_READY] } - { [BOOL_UP_MOVE] | [BOOL_DOWN_MOVE] }
		EN --- MOVE(UINT_UD_ACCDCC) => ACC_UINT
		EN --- MOVE(UINT_UD_ACCDCC) => DCC_UINT
NETWORK 10
	[BOOL_UP_MOVE] - T1:TON(IN: *, PT: TIME_UD_DLY_ON, ET => T1COUNT) --- (UP_MOVE_ST_BOOL)
NETWORK 11
	[BOOL_DOWN_MOVE] - T2:TON(IN: *, PT: TIME_UD_DLY_ON, ET => T2COUNT) --- (DOWN_MOVE_ST_BOOL)
_END_LD_
(* the same logic as Structured Text *)
(* Network 1 *)
MANJOGH := STRING_CURRENT_PG = STRING_MAN_JOG_H_PG;
(* Network 2 *)
MANJOGV := STRING_CURRENT_PG = STRING_MAN_JOG_V_PG;
(* Network 3 *)
MANPOSH := STRING_CURRENT_PG = STRING_MAN_POS_H_PG;
(* Network 4 *)
MANPOSV := STRING_CURRENT_PG = STRING_MAN_POS_V_PG;
(* Network 5 *)
(* Network 6 *)
IF MANJOGH OR MANJOGV THEN
	ACC_UINT := UINT_JOG_ACCDCC;
	DCC_UINT := UINT_JOG_ACCDCC;
END_IF;
(* Network 7 *)
IF NOT BOOL_MANUAL_PG AND NOT BOOL_ORIGIN_COMP OR (MANPOSH OR MANPOSV) AND BOOL_MANUAL_PG AND NOT BOOL_ARM_HOME_READY THEN
	ACC_UINT := UINT_HOME_ACCDCC;
	DCC_UINT := UINT_HOME_ACCDCC;
END_IF;
(* Network 8 *)
IF (BOOL_ORIGIN_COMP OR (MANPOSH OR MANPOSV) AND BOOL_MANUAL_PG AND BOOL_ARM_HOME_READY) AND NOT BOOL_UP_MOVE AND NOT BOOL_DOWN_MOVE THEN
	ACC_UINT := UINT_AG_ACCDCC;
	DCC_UINT := UINT_AG_ACCDCC;
END_IF;
(* Network 9 *)
IF (BOOL_ORIGIN_COMP OR (MANPOSH OR MANPOSV) AND BOOL_MANUAL_PG AND BOOL_ARM_HOME_READY) AND (BOOL_UP_MOVE OR BOOL_DOWN_MOVE) THEN
	ACC_UINT := UINT_UD_ACCDCC;
	DCC_UINT := UINT_UD_ACCDCC;
END_IF;
(* Network 10 *)
T1(IN := BOOL_UP_MOVE, PT := TIME_UD_DLY_ON);
T1COUNT := T1.ET;
UP_MOVE_ST_BOOL := T1.Q;
(* Network 11 *)
T2(IN := BOOL_DOWN_MOVE, PT := TIME_UD_DLY_ON);
T2COUNT := T2.ET;
DOWN_MOVE_ST_BOOL := T2.Q;
END_FUNCTION_BLOCK

(* POU MOTION_COUNTER_RESET, LD *)
FUNCTION_BLOCK MOTION_COUNTER_RESET
VAR_INPUT
	BOOL_JOG_ACTIVE : BOOL;
	TIME_RST_DELAY_OFF : TIME;
END_VAR
VAR_OUTPUT
	COUNTER_RST_BOOL : BOOL;
END_VAR
VAR
	DFN: F_TRIG;
	JOGDFN: BOOL;
	T1: TON;
	T1ON: BOOL;
	t0: TON;
	CUTDELAY: BOOL;
END_VAR
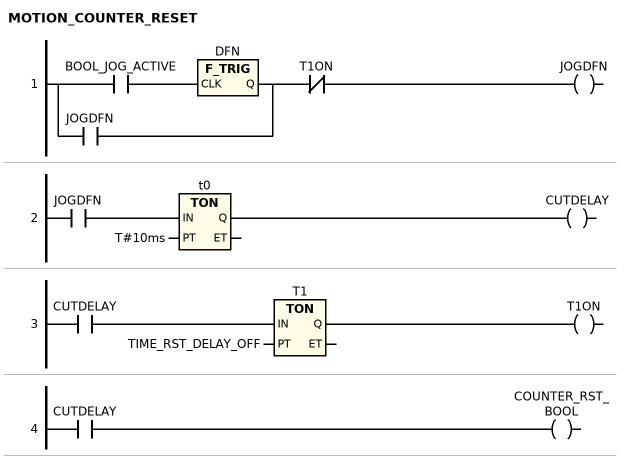
_LD_ (* Ladder Diagram *)
NETWORK 1
	{ [BOOL_JOG_ACTIVE] - DFN:F_TRIG(CLK: *) | [JOGDFN] } - [/T1ON] --- (JOGDFN)
NETWORK 2
	[JOGDFN] - t0:TON(IN: *, PT: T#10ms) --- (CUTDELAY)
NETWORK 3
	[CUTDELAY] - T1:TON(IN: *, PT: TIME_RST_DELAY_OFF) --- (T1ON)
NETWORK 4
	[CUTDELAY] --- (COUNTER_RST_BOOL)
_END_LD_
(* the same logic as Structured Text *)
(* Network 1 *)
DFN(CLK := BOOL_JOG_ACTIVE);
JOGDFN := (DFN.Q OR JOGDFN) AND NOT T1ON;
(* Network 2 *)
t0(IN := JOGDFN, PT := T#10ms);
CUTDELAY := t0.Q;
(* Network 3 *)
T1(IN := CUTDELAY, PT := TIME_RST_DELAY_OFF);
T1ON := T1.Q;
(* Network 4 *)
COUNTER_RST_BOOL := CUTDELAY;
END_FUNCTION_BLOCK

(* POU MUL_ARM_BASKET_MEMORY, LD *)
FUNCTION_BLOCK MUL_ARM_BASKET_MEMORY
VAR_INPUT
	bLoadUnhook:BOOL;
	bLoadHook:BOOL;
	bUnloadUnhook: BOOL;
	bUnloadHook:BOOL;
	bArmDown: BOOL;
	tSignalFilter : TIME;

END_VAR

VAR_OUTPUT
(*	bPreviousZoneSensor2On: BOOL;
	bPreviousZoneSensor1On: BOOL;
	Inhibit: BOOL;*)


	bNoCurrentStationConfirmBasketFlag: BOOL;
	bNoCurrentStationTransferBasketFlag: BOOL;
	bNoNextStationConfirmBasketFlag: BOOL;
END_VAR
VAR

	LoadUnhookConfirmTimer: TON;
	LoadHookConfirmTimer: TON;
	UnloadUnhookConfirmTimer: TON;
	UnloadHookConfirmTimer: TON;
	PowerUpDelayTimer: TON;
	PUDT_Out: BOOL;


	LoadUnhookDIFU: R_TRIG;
	LoadHookDIFU: R_TRIG;
	UnloadUnhookDIFU: R_TRIG;
	UnloadHookDIFU: R_TRIG;
END_VAR
VAR_IN_OUT


	CurrentStationConfirmBasketName:STRING;
	CurrentStationTransferBasketName:STRING;
	NextStationConfirmBasketName:STRING;

END_VAR
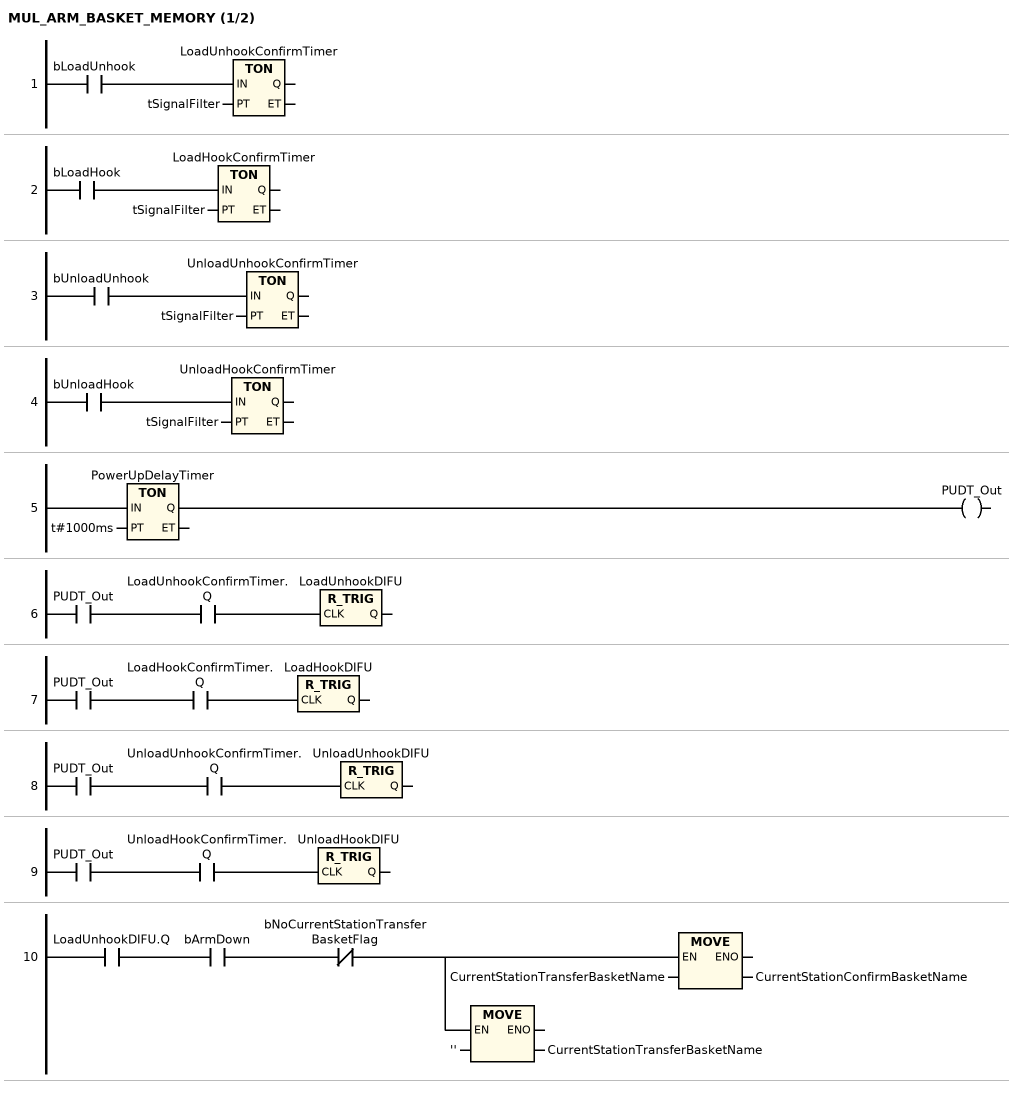
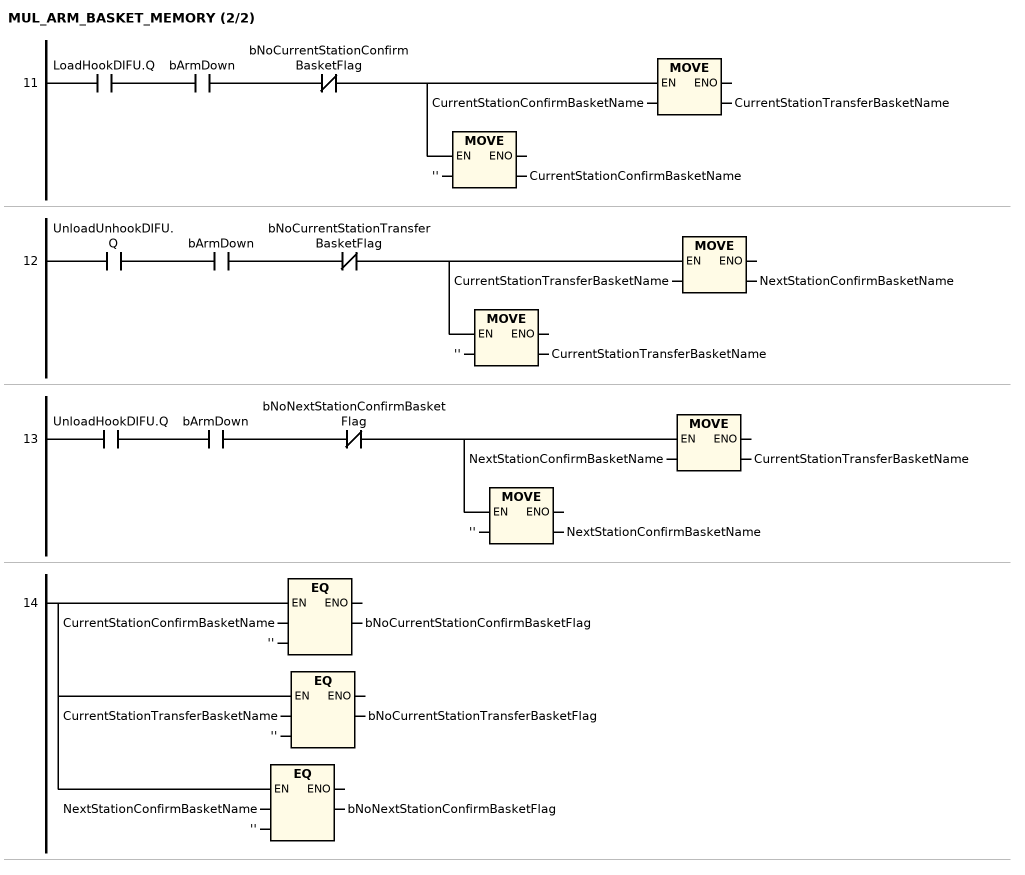
_LD_ (* Ladder Diagram *)
NETWORK 1
	[bLoadUnhook] - LoadUnhookConfirmTimer:TON(IN: *, PT: tSignalFilter)
NETWORK 2
	[bLoadHook] - LoadHookConfirmTimer:TON(IN: *, PT: tSignalFilter)
NETWORK 3
	[bUnloadUnhook] - UnloadUnhookConfirmTimer:TON(IN: *, PT: tSignalFilter)
NETWORK 4
	[bUnloadHook] - UnloadHookConfirmTimer:TON(IN: *, PT: tSignalFilter)
NETWORK 5
	PowerUpDelayTimer:TON(IN: *, PT: t#1000ms) --- (PUDT_Out)
NETWORK 6
	[PUDT_Out] - [LoadUnhookConfirmTimer.Q] - LoadUnhookDIFU:R_TRIG(CLK: *)
NETWORK 7
	[PUDT_Out] - [LoadHookConfirmTimer.Q] - LoadHookDIFU:R_TRIG(CLK: *)
NETWORK 8
	[PUDT_Out] - [UnloadUnhookConfirmTimer.Q] - UnloadUnhookDIFU:R_TRIG(CLK: *)
NETWORK 9
	[PUDT_Out] - [UnloadHookConfirmTimer.Q] - UnloadHookDIFU:R_TRIG(CLK: *)
NETWORK 10
	[LoadUnhookDIFU.Q] - [bArmDown] - [/bNoCurrentStationTransferBasketFlag]
		EN --- MOVE(CurrentStationTransferBasketName) => CurrentStationConfirmBasketName
		EN --- MOVE('') => CurrentStationTransferBasketName
NETWORK 11
	[LoadHookDIFU.Q] - [bArmDown] - [/bNoCurrentStationConfirmBasketFlag]
		EN --- MOVE(CurrentStationConfirmBasketName) => CurrentStationTransferBasketName
		EN --- MOVE('') => CurrentStationConfirmBasketName
NETWORK 12
	[UnloadUnhookDIFU.Q] - [bArmDown] - [/bNoCurrentStationTransferBasketFlag]
		EN --- MOVE(CurrentStationTransferBasketName) => NextStationConfirmBasketName
		EN --- MOVE('') => CurrentStationTransferBasketName
NETWORK 13
	[UnloadHookDIFU.Q] - [bArmDown] - [/bNoNextStationConfirmBasketFlag]
		EN --- MOVE(NextStationConfirmBasketName) => CurrentStationTransferBasketName
		EN --- MOVE('') => NextStationConfirmBasketName
NETWORK 14
	*
		EN --- EQ(CurrentStationConfirmBasketName, '') => bNoCurrentStationConfirmBasketFlag
		EN --- EQ(CurrentStationTransferBasketName, '') => bNoCurrentStationTransferBasketFlag
		EN --- EQ(NextStationConfirmBasketName, '') => bNoNextStationConfirmBasketFlag
_END_LD_
(* the same logic as Structured Text *)
(* Network 1 *)
LoadUnhookConfirmTimer(IN := bLoadUnhook, PT := tSignalFilter);
(* Network 2 *)
LoadHookConfirmTimer(IN := bLoadHook, PT := tSignalFilter);
(* Network 3 *)
UnloadUnhookConfirmTimer(IN := bUnloadUnhook, PT := tSignalFilter);
(* Network 4 *)
UnloadHookConfirmTimer(IN := bUnloadHook, PT := tSignalFilter);
(* Network 5 *)
PowerUpDelayTimer(IN := TRUE, PT := t#1000ms);
PUDT_Out := PowerUpDelayTimer.Q;
(* Network 6 *)
LoadUnhookDIFU(CLK := PUDT_Out AND LoadUnhookConfirmTimer.Q);
(* Network 7 *)
LoadHookDIFU(CLK := PUDT_Out AND LoadHookConfirmTimer.Q);
(* Network 8 *)
UnloadUnhookDIFU(CLK := PUDT_Out AND UnloadUnhookConfirmTimer.Q);
(* Network 9 *)
UnloadHookDIFU(CLK := PUDT_Out AND UnloadHookConfirmTimer.Q);
(* Network 10 *)
IF LoadUnhookDIFU.Q AND bArmDown AND NOT bNoCurrentStationTransferBasketFlag THEN
	CurrentStationConfirmBasketName := CurrentStationTransferBasketName;
	CurrentStationTransferBasketName := '';
END_IF;
(* Network 11 *)
IF LoadHookDIFU.Q AND bArmDown AND NOT bNoCurrentStationConfirmBasketFlag THEN
	CurrentStationTransferBasketName := CurrentStationConfirmBasketName;
	CurrentStationConfirmBasketName := '';
END_IF;
(* Network 12 *)
IF UnloadUnhookDIFU.Q AND bArmDown AND NOT bNoCurrentStationTransferBasketFlag THEN
	NextStationConfirmBasketName := CurrentStationTransferBasketName;
	CurrentStationTransferBasketName := '';
END_IF;
(* Network 13 *)
IF UnloadHookDIFU.Q AND bArmDown AND NOT bNoNextStationConfirmBasketFlag THEN
	CurrentStationTransferBasketName := NextStationConfirmBasketName;
	NextStationConfirmBasketName := '';
END_IF;
(* Network 14 *)
bNoCurrentStationConfirmBasketFlag := CurrentStationConfirmBasketName = '';
bNoCurrentStationTransferBasketFlag := CurrentStationTransferBasketName = '';
bNoNextStationConfirmBasketFlag := NextStationConfirmBasketName = '';
END_FUNCTION_BLOCK

(* POU SERVO_POS_CONFIRM, LD *)
FUNCTION_BLOCK SERVO_POS_CONFIRM
VAR_INPUT
	BOOL_JOG_ACTIVE : BOOL;
	UINT_TARGET1 : UINT;
	UINT_TARGET2 : UINT;
	UINT_TARGET3 : UINT;
	UINT_TARGET4 : UINT;
	COUNTER_VALUE : UINT;
	HOMING_READY : BOOL;
END_VAR

VAR_OUTPUT
	TARGET1_CONFIRM_BOOL : BOOL;
	TARGET2_CONFIRM_BOOL : BOOL;
	TARGET3_CONFIRM_BOOL : BOOL;
	TARGET4_CONFIRM_BOOL : BOOL;
END_VAR
VAR
	T1C: BOOL;
	T2C: BOOL;
	T3C: BOOL;
	T4C: BOOL;
END_VAR
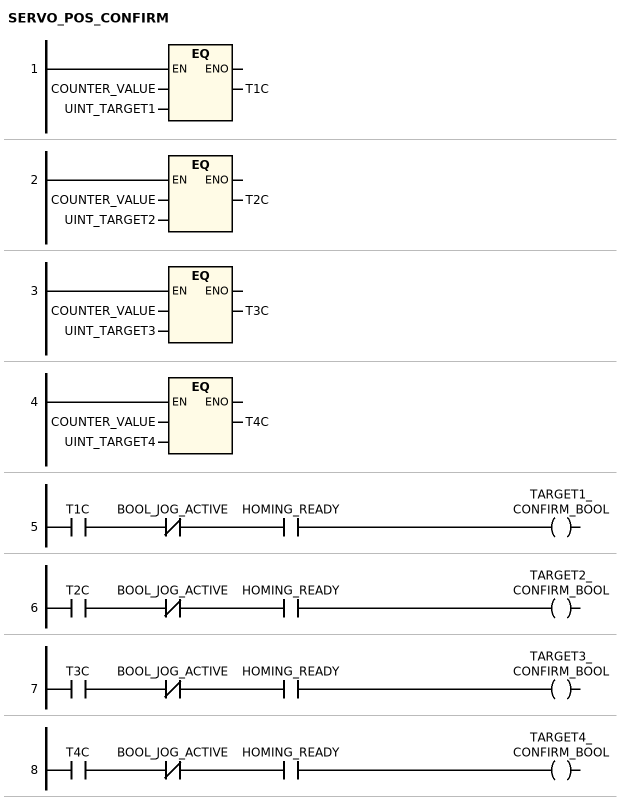
_LD_ (* Ladder Diagram *)
NETWORK 1
	*
		EN --- EQ(COUNTER_VALUE, UINT_TARGET1) => T1C
NETWORK 2
	*
		EN --- EQ(COUNTER_VALUE, UINT_TARGET2) => T2C
NETWORK 3
	*
		EN --- EQ(COUNTER_VALUE, UINT_TARGET3) => T3C
NETWORK 4
	*
		EN --- EQ(COUNTER_VALUE, UINT_TARGET4) => T4C
NETWORK 5
	[T1C] - [/BOOL_JOG_ACTIVE] - [HOMING_READY] --- (TARGET1_CONFIRM_BOOL)
NETWORK 6
	[T2C] - [/BOOL_JOG_ACTIVE] - [HOMING_READY] --- (TARGET2_CONFIRM_BOOL)
NETWORK 7
	[T3C] - [/BOOL_JOG_ACTIVE] - [HOMING_READY] --- (TARGET3_CONFIRM_BOOL)
NETWORK 8
	[T4C] - [/BOOL_JOG_ACTIVE] - [HOMING_READY] --- (TARGET4_CONFIRM_BOOL)
_END_LD_
(* the same logic as Structured Text *)
(* Network 1 *)
T1C := COUNTER_VALUE = UINT_TARGET1;
(* Network 2 *)
T2C := COUNTER_VALUE = UINT_TARGET2;
(* Network 3 *)
T3C := COUNTER_VALUE = UINT_TARGET3;
(* Network 4 *)
T4C := COUNTER_VALUE = UINT_TARGET4;
(* Network 5 *)
TARGET1_CONFIRM_BOOL := T1C AND NOT BOOL_JOG_ACTIVE AND HOMING_READY;
(* Network 6 *)
TARGET2_CONFIRM_BOOL := T2C AND NOT BOOL_JOG_ACTIVE AND HOMING_READY;
(* Network 7 *)
TARGET3_CONFIRM_BOOL := T3C AND NOT BOOL_JOG_ACTIVE AND HOMING_READY;
(* Network 8 *)
TARGET4_CONFIRM_BOOL := T4C AND NOT BOOL_JOG_ACTIVE AND HOMING_READY;
END_FUNCTION_BLOCK

(* POU TEMP_CTRL_ON_OFF, FBD *)
FUNCTION_BLOCK TEMP_CTRL_ON_OFF
VAR_INPUT
	REAL_SV			: REAL;
	REAL_HYS			: REAL;
	REAL_HAL			: REAL;
	REAL_T_READY		: REAL; (*Value set base on -X*)
END_VAR


VAR_OUTPUT
	REAL_PV : REAL;
	OUT_BOOL: BOOL;
	HAL_BOOL: BOOL;
	T_READY_BOOL: BOOL;

END_VAR
VAR
	TEMP_PV	AT %I*	: INT;
	TREADY_TEMP: REAL;
	HYS_TEMP: REAL;
	ALWAYS_OFF: BOOL;
	ALWAYS_ON_BOOL: BOOL;
	T1: TON;
	PLS1: R_TRIG;
	RS1: RS;
END_VAR
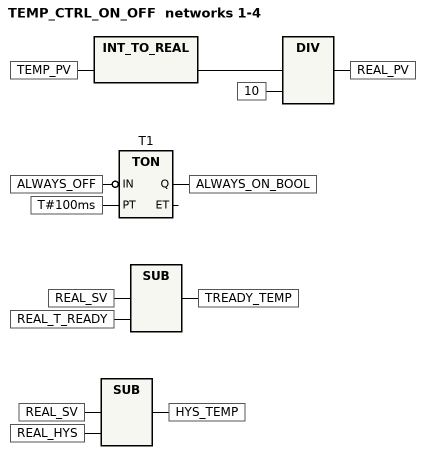
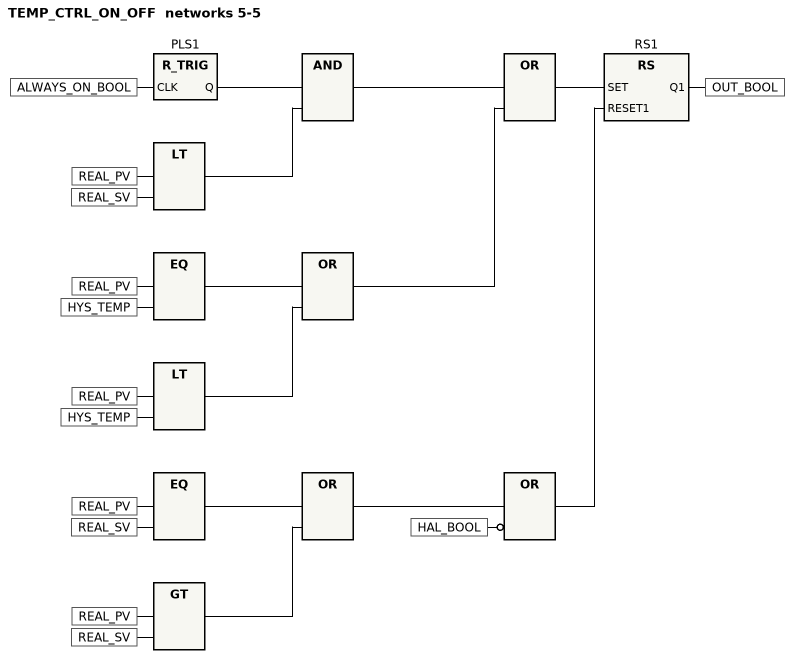
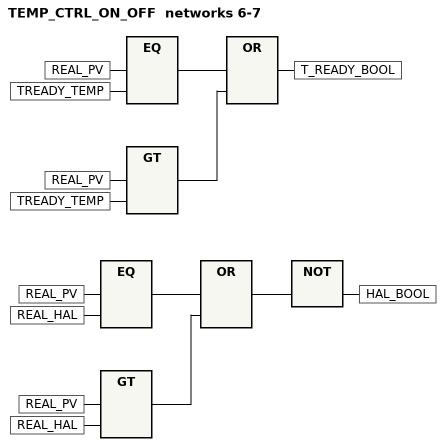
_FBD_ (* Function Block Diagram *)
NETWORK 1
	DIV(INT_TO_REAL(TEMP_PV), 10) => REAL_PV
NETWORK 2
	T1:TON(IN: NOT ALWAYS_OFF, PT: T#100ms) => ALWAYS_ON_BOOL
NETWORK 3
	SUB(REAL_SV, REAL_T_READY) => TREADY_TEMP
NETWORK 4
	SUB(REAL_SV, REAL_HYS) => HYS_TEMP
NETWORK 5
	RS1:RS(SET: OR(AND(PLS1:R_TRIG(CLK: ALWAYS_ON_BOOL), LT(REAL_PV, REAL_SV)), OR(EQ(REAL_PV, HYS_TEMP), LT(REAL_PV, HYS_TEMP))), RESET1: OR(OR(EQ(REAL_PV, REAL_SV), GT(REAL_PV, REAL_SV)), NOT HAL_BOOL)) => OUT_BOOL
NETWORK 6
	OR(EQ(REAL_PV, TREADY_TEMP), GT(REAL_PV, TREADY_TEMP)) => T_READY_BOOL
NETWORK 7
	NOT OR(EQ(REAL_PV, REAL_HAL), GT(REAL_PV, REAL_HAL)) => HAL_BOOL
_END_FBD_
(* the same logic as Structured Text *)
(* Network 1 *)
REAL_PV := INT_TO_REAL(TEMP_PV) / 10;
(* Network 2 *)
T1(IN := NOT ALWAYS_OFF, PT := T#100ms);
ALWAYS_ON_BOOL := T1.Q;
(* Network 3 *)
TREADY_TEMP := REAL_SV - REAL_T_READY;
(* Network 4 *)
HYS_TEMP := REAL_SV - REAL_HYS;
(* Network 5 *)
PLS1(CLK := ALWAYS_ON_BOOL);
RS1(SET := (PLS1.Q AND (REAL_PV < REAL_SV)) OR ((REAL_PV = HYS_TEMP) OR (REAL_PV < HYS_TEMP)), RESET1 := ((REAL_PV = REAL_SV) OR (REAL_PV > REAL_SV)) OR NOT HAL_BOOL);
OUT_BOOL := RS1.Q1;
(* Network 6 *)
T_READY_BOOL := (REAL_PV = TREADY_TEMP) OR (REAL_PV > TREADY_TEMP);
(* Network 7 *)
HAL_BOOL := NOT ((REAL_PV = REAL_HAL) OR (REAL_PV > REAL_HAL));
END_FUNCTION_BLOCK

(* POU TIMER_ALARM, LD *)
FUNCTION_BLOCK TIMER_ALARM
VAR_INPUT
	BOOL_SIGNAL_IN: BOOL;
	BOOL_ALMRST_PB: BOOL;
	BOOL_BZRST_PB: BOOL;
	INT_PV: INT;

END_VAR

VAR_OUTPUT
	ALM_MSG_BOOL: BOOL;
	BZ_OUT_BOOL: BOOL;
	EV_INT: INT;
END_VAR

VAR
	T1: TON;
	M0: BOOL;
	M1: BOOL;
	D200: TIME;
	D202: INT;
END_VAR
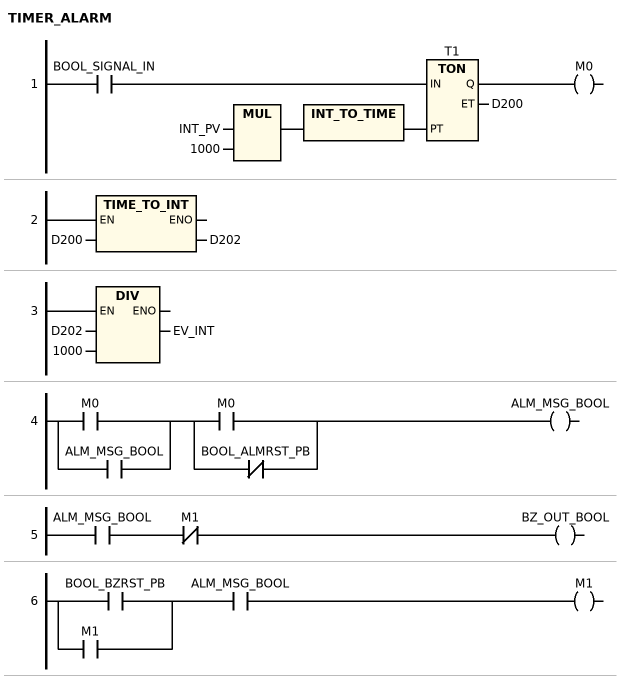
_LD_ (* Ladder Diagram *)
NETWORK 1
	[BOOL_SIGNAL_IN] - T1:TON(IN: *, PT: INT_TO_TIME(MUL(INT_PV, 1000)), ET => D200) --- (M0)
NETWORK 2
	*
		EN --- TIME_TO_INT(D200) => D202
NETWORK 3
	*
		EN --- DIV(D202, 1000) => EV_INT
NETWORK 4
	{ [M0] | [ALM_MSG_BOOL] } - { [M0] | [/BOOL_ALMRST_PB] } --- (ALM_MSG_BOOL)
NETWORK 5
	[ALM_MSG_BOOL] - [/M1] --- (BZ_OUT_BOOL)
NETWORK 6
	{ [BOOL_BZRST_PB] | [M1] } - [ALM_MSG_BOOL] --- (M1)
_END_LD_
(* the same logic as Structured Text *)
(* Network 1 *)
T1(IN := BOOL_SIGNAL_IN, PT := INT_TO_TIME(INT_PV * 1000));
D200 := T1.ET;
M0 := T1.Q;
(* Network 2 *)
D202 := TIME_TO_INT(D200);
(* Network 3 *)
EV_INT := D202 / 1000;
(* Network 4 *)
ALM_MSG_BOOL := (M0 OR ALM_MSG_BOOL) AND (M0 OR NOT BOOL_ALMRST_PB);
(* Network 5 *)
BZ_OUT_BOOL := ALM_MSG_BOOL AND NOT M1;
(* Network 6 *)
M1 := (BOOL_BZRST_PB OR M1) AND ALM_MSG_BOOL;
END_FUNCTION_BLOCK
